(* ========================================================= *)
(*    FUN: HLI_ChannelModeReference                          *)
(* --------------------------------------------------------- *)
(*   Desc: switch channel to Reference mode / xxx            *)
(*   Author: MK, MiB, TV                                     *)
(*   Date: 03.03.2017                                        *)
(*   Rev.: 1.5                                               *)
(* ========================================================= *)


(************************************************************
	RefPosString:
	Element: parameter ( ASCII char set, Länge:256 Zeichen)

	Vorgabe zur Parametrierung der Referenzpunktfahrt.

	Ist dieser STRING leer, so wird defaultmäßig das
	Automatikprogramm "rpf.nc" angewählt.

	Ansonsten kann durch explizite Angabe der Achsen und
	Zeitpunkt im Format "G74
	<Achsbezeichner_1><Zeitpunkt_1> ...
	<Achsbezeichner_n><Zeitpunkt_n>"
	eine individuelle Referenzpunktfahrt vorgegeben werden.
*************************************************************)

IF (NOT gpCh[nChanIdx]^.channel_mc_control.mode_and_state.command_semaphor_rw) THEN  (* only if semaphor is FALSE...... *)
	IF stCmdModesStates.stStates.Selected THEN
		stCmdModesStates.stStates.Selected := FALSE;
		gpCh[nChanIdx]^.channel_mc_control.mode_and_state.command_w.to_mode := HLI_IMCM_REFERENCE_MODE;
		gpCh[nChanIdx]^.channel_mc_control.mode_and_state.command_w.to_state := HLI_IMCM_PROCESS_SELECTED;		
		gpCh[nChanIdx]^.channel_mc_control.mode_and_state.command_semaphor_rw := TRUE;	
	END_IF
	
	IF stCmdModesStates.stStates.Ready THEN
		stCmdModesStates.stStates.Ready := FALSE;
		gpCh[nChanIdx]^.channel_mc_control.mode_and_state.command_w.to_mode := HLI_IMCM_REFERENCE_MODE;
		gpCh[nChanIdx]^.channel_mc_control.mode_and_state.command_w.to_state := HLI_IMCM_PROCESS_READY;		
		pString := ADR(gpCh[nChanIdx]^.channel_mc_control.mode_and_state.command_w.parameter);	
		gpCh[nChanIdx]^.channel_mc_control.mode_and_state.command_semaphor_rw := TRUE;		
	END_IF
	
	IF stCmdModesStates.stStates.Active THEN
		stCmdModesStates.stStates.Active := FALSE;
		gpCh[nChanIdx]^.channel_mc_control.mode_and_state.command_w.to_mode := HLI_IMCM_REFERENCE_MODE;
		gpCh[nChanIdx]^.channel_mc_control.mode_and_state.command_w.to_state := HLI_IMCM_PROCESS_ACTIVE;		
		pString := ADR(gpCh[nChanIdx]^.channel_mc_control.mode_and_state.command_w.parameter);	
		pString^ := sRefPosString;
		gpCh[nChanIdx]^.channel_mc_control.mode_and_state.command_semaphor_rw:= TRUE;		
	END_IF
	
	IF stCmdModesStates.stStates.Hold THEN
		stCmdModesStates.stStates.Hold := FALSE;
		gpCh[nChanIdx]^.channel_mc_control.mode_and_state.command_w.to_mode := HLI_IMCM_REFERENCE_MODE;
		gpCh[nChanIdx]^.channel_mc_control.mode_and_state.command_w.to_state := HLI_IMCM_PROCESS_HOLD;		
		gpCh[nChanIdx]^.channel_mc_control.mode_and_state.command_semaphor_rw := TRUE;		
	END_IF
	
	IF stCmdModesStates.stStates.Reset THEN
		stCmdModesStates.stStates.Reset := FALSE;
		gpCh[nChanIdx]^.channel_mc_control.mode_and_state.command_w.to_mode:= HLI_IMCM_REFERENCE_MODE;
		gpCh[nChanIdx]^.channel_mc_control.mode_and_state.command_w.to_state := HLI_IMCM_PROCESS_DESELECTED;		
		gpCh[nChanIdx]^.channel_mc_control.mode_and_state.command_semaphor_rw := TRUE;		
	END_IF

	HLI3_ChannelModeReference := TRUE;
ELSE
	HLI3_ChannelModeReference := FALSE;
END_IF

END_FUNCTION

// CNC/2 OperationMode/HLI3_ChannelModeStandby
FUNCTION HLI3_ChannelModeStandby : BOOL
VAR_INPUT	 
	nChanIdx: INT;
	ProgramName: STRING(HLI_IMCM_MODE_STATE_PARAM_STRL);			
END_VAR

VAR_IN_OUT
	stCmdModesStates    : ST_CNCCmdModesStates;	
END_VAR

VAR
	pString: POINTER TO STRING(HLI_IMCM_MODE_STATE_PARAM_STRL);
	nCHan: INT;
END_VAR

(* ========================================================= *)
(*    FUN: HLI_ChannelModeStandby                            *)
(* --------------------------------------------------------- *)
(*   Desc: switch channel to Standby mode / xxx              *)
(*   Author: MK, MiB, TV                                     *)
(*   Date: 03.03.2017                                        *)
(*   Rev.: 1.5                                               *)
(* ========================================================= *)

IF (NOT gpCh[nChanIdx]^.channel_mc_control.mode_and_state.command_semaphor_rw) THEN  (* only if semaphor is FALSE...... *)
	IF stCmdModesStates.stStates.Selected THEN
		stCmdModesStates.stStates.Selected := FALSE;
		gpCh[nChanIdx]^.channel_mc_control.mode_and_state.command_w.to_mode := HLI_IMCM_STANDBY_MODE;
		gpCh[nChanIdx]^.channel_mc_control.mode_and_state.command_w.to_state := HLI_IMCM_PROCESS_SELECTED;
		pString := ADR(gpCh[nChanIdx]^.channel_mc_control.mode_and_state.command_w.parameter);			
		pString^ := ProgramName;				
		gpCh[nChanIdx]^.channel_mc_control.mode_and_state.command_semaphor_rw := TRUE;		
	END_IF
	
	IF stCmdModesStates.stStates.Ready THEN
		stCmdModesStates.stStates.Ready := FALSE;
		gpCh[nChanIdx]^.channel_mc_control.mode_and_state.command_w.to_mode := HLI_IMCM_STANDBY_MODE;
		gpCh[nChanIdx]^.channel_mc_control.mode_and_state.command_w.to_state := HLI_IMCM_PROCESS_READY;		
		pString := ADR(gpCh[nChanIdx]^.channel_mc_control.mode_and_state.command_w.parameter);			
		pString^ := ProgramName;	
		gpCh[nChanIdx]^.channel_mc_control.mode_and_state.command_semaphor_rw := TRUE;		
	END_IF
	
	IF stCmdModesStates.stStates.Active THEN
		stCmdModesStates.stStates.Active := FALSE;
		gpCh[nChanIdx]^.channel_mc_control.mode_and_state.command_w.to_mode := HLI_IMCM_STANDBY_MODE;
		gpCh[nChanIdx]^.channel_mc_control.mode_and_state.command_w.to_state := HLI_IMCM_PROCESS_ACTIVE;		
		pString := ADR(gpCh[nChanIdx]^.channel_mc_control.mode_and_state.command_w.parameter);			
		pString^ := ProgramName;	
		gpCh[nChanIdx]^.channel_mc_control.mode_and_state.command_semaphor_rw := TRUE;		
	END_IF
	
	IF stCmdModesStates.stStates.Hold THEN
		stCmdModesStates.stStates.Hold := FALSE;
		gpCh[nChanIdx]^.channel_mc_control.mode_and_state.command_w.to_mode := HLI_IMCM_STANDBY_MODE;
		gpCh[nChanIdx]^.channel_mc_control.mode_and_state.command_w.to_state:= HLI_IMCM_PROCESS_HOLD;		
		gpCh[nChanIdx]^.channel_mc_control.mode_and_state.command_semaphor_rw := TRUE;	
	END_IF
	
	IF stCmdModesStates.stStates.Reset THEN
		stCmdModesStates.stStates.Reset := FALSE;
		gpCh[nChanIdx]^.channel_mc_control.mode_and_state.command_w.to_mode := HLI_IMCM_STANDBY_MODE;
		gpCh[nChanIdx]^.channel_mc_control.mode_and_state.command_w.to_state:= HLI_IMCM_PROCESS_DESELECTED;		
		gpCh[nChanIdx]^.channel_mc_control.mode_and_state.command_semaphor_rw := TRUE;		
	END_IF
	
	HLI3_ChannelModeStandby := TRUE;
ELSE
	HLI3_ChannelModeStandby := FALSE;
END_IF

END_FUNCTION

// CNC/2 OperationMode/HLI3_ChannelReset
FUNCTION HLI3_ChannelReset : BOOL
VAR_INPUT
	/// Channel index 
	nChanIdx: INT;
END_VAR
VAR
	/// local pointer to Data of actual Channel 
	pChannelData: POINTER TO HIGH_LEVEL_INTERFACE_CH;
END_VAR

(* ========================================================= *)
(*    FUN: HLI_ChannelReset                                  *)
(* --------------------------------------------------------- *)
(*   Desc:                                                   *)
(* Author: MK ,MiB, TV                                       *)
(*   Date: 17.01.2018                                        *)
(*   Rev.: 1.1                                               *)
(* ========================================================= *)

HLI3_ChannelReset := FALSE;
IF NOT HLI3_CheckChannelValid(nChannel := nChanIdx) THEN
	RETURN;
END_IF

(* get pointer to channel data *)
pChannelData := gpCh[nChanIdx];
IF (pChannelData = 0) THEN   (* check for zero pointer *)
	RETURN;
END_IF

(* is a reset commanded *)
IF pChannelData^.bahn_lc_control.plc_reset.command_r = TRUE THEN
	
(* Reset all M- and H-Functions whenn the channel gets resetted *)
	HLI3_ChannelResetMFunctions(nChanIdx);
	HLI3_ChannelResetHFunctions(nChanIdx);
	
	(* quit this reset *)
	pChannelData^.bahn_lc_control.plc_reset.state_w := TRUE;	
	HLI3_ChannelReset := TRUE;
END_IF

END_FUNCTION

// CNC/4 MHT-Function/HLI3_ChannelResetMFunctions
FUNCTION HLI3_ChannelResetMFunctions : BOOL
VAR_INPUT
	/// Channel number 
	nChanIdx: INT;
END_VAR
VAR
	idx: INT;
END_VAR

(* ========================================================= *)
(*    FUN: HLI_ChannelResetMFunctions                        *)
(* --------------------------------------------------------- *)
(*   Desc:                                                   *)
(* Author: MK                                                *)
(*   Date: 10.05.2007                                        *)
(*   Rev.: 1.00                                              *)
(* ========================================================= *)

IF NOT HLI3_CheckChannelValid(nChannel := nChanIdx) THEN
	HLI3_ChannelResetMFunctions := FALSE;
	RETURN; (* A b b r u c h *)
END_IF


FOR idx := 1 TO 999 DO
	CNCSystem.Channel[nChanIdx].M[idx].bState_rw := FALSE;
	CNCSystem.Channel[nChanIdx].M[idx].bRes := FALSE;
	CNCSystem.Channel[nChanIdx].actM_r :='';
END_FOR

HLI3_ChannelResetMFunctions := TRUE;

END_FUNCTION

// CNC/4 MHT-Function/HLI3_ChannelResetHFunctions
FUNCTION HLI3_ChannelResetHFunctions : BOOL
VAR_INPUT
	/// Channel number 
	nChanIdx: INT;
END_VAR
VAR
	idx: INT;
END_VAR

(* ========================================================= *)
(*    FUN: HLI_ChannelResetHFunctions                        *)
(* --------------------------------------------------------- *)
(*   Desc:                                                   *)
(* Author: MiB                                                *)
(*   Date: 23.11.2012                                        *)
(*   Rev.: 1.1                                              *)
(* ========================================================= *)



IF NOT HLI3_CheckChannelValid(nChannel := nChanIdx) THEN
	HLI3_ChannelResetHFunctions := FALSE;
	RETURN; (* A b b r u c h *)
END_IF


FOR idx := 0 TO 999 DO
	CNCSystem.Channel[nChanIdx].H[idx].bState_rw := FALSE;
	CNCSystem.Channel[nChanIdx].H[idx].bRes := FALSE;
	CNCSystem.Channel[nChanIdx].actH_r :='';
END_FOR

HLI3_ChannelResetHFunctions := TRUE;

END_FUNCTION

// CNC/2 OperationMode/HLI3_ChannelResetRequest
FUNCTION_BLOCK HLI3_ChannelResetRequest
VAR_INPUT
	bExec: BOOL;
	/// Channel number 
	nChanIdx: INT;
	pChannel: POINTER TO ST_CncChannel;
END_VAR
VAR_OUTPUT
	bBusy: BOOL;
	bSwitchMode: BOOL;
	nMode: UDINT;
END_VAR
VAR
	fbRtrigExec: R_TRIG;
	/// Index of channel specific HLI area 
	nHliChIfcIdx: INT;
	nState: UINT;
	pCommand: POINTER TO HLI_PROC_TRANS_TO_MODE_STATE;
	actualMode: UDINT;
	fbTON: TON;
END_VAR

(******************************************************************************)
(* POU:				HLI_ChannelResetRequest									*)
(* Type:				Function block										*)
(* Customer:		Common													*)
(* Date:				07/11/16											*)
(* Last:				10/03/10											*)
(* -------------------------------------------------------------------------- *)
(* Revision:		1.0														*)
(* Author:			MiB														*)
(* Description: 	Performs a reset in the given cnc channel. 				*)
(* -------------------------------------------------------------------------- *)
(* Revision:		1.10													*)
(* Author:			MiB														*)
(* Description: 	Changed from PRG to FB.									*)
(* -------------------------------------------------------------------------- *)
(* Revision:		2.00															*)
(* Author:			HR																*)
(* Description: 	Deleted references to global variable 'PLCMachineMode[n]'.		*)
(*						The FB now works with VAR_OUTPUT 'nMode' and 'bSwitchMode'	*)
(*						as a callback to the initiator to let it perform the change	*)
(*						of the operation mode by itself in order to reset the cnc	*)
(*						channel.													*)
(* -------------------------------------------------------------------------- *)
(* Revision:		2.01																			*)
(* Author:			TV																				*)
(* Description: 	Expand State "Wait for previous mode"  *)
(*				Prevent to trigger the state machine during the mode switch							*)
(* -------------------------------------------------------------------------- *)
(* Revision:		2.02																			*)
(* Author:			MiB																				*)
(* Description: 	Tc3*)
(******************************************************************************)


fbRtrigExec( clk := bExec   );

IF fbRtrigExec.Q THEN
	bBusy := TRUE;
	nState := 10;
END_IF


CASE nState OF

0:		(* IDLE *)
		bBusy := FALSE;

10:	(* Reset request: get actual opmode *)
		bSwitchMode := FALSE;
		actualMode := gpCh[nChanIdx]^.channel_mc_control.mode_and_state.state_r.mode;
		nState := nState + 10;

20:  (* switch to standby *)
		bSwitchMode := TRUE;
		nMode:= HLI_IMCM_STANDBY_MODE;
		fbTON(IN:= FALSE);
		nState := nState + 10;

30: 	(* Wait for modeswitch *)
		bSwitchMode := FALSE;
		fbTON(IN:= TRUE, PT:= t#2000ms);
	 	IF gpCh[nChanIdx]^.channel_mc_control.mode_and_state.state_r.mode = HLI_IMCM_STANDBY_MODE THEN
			nState := nState + 10;
		END_IF
		IF fbTON.Q THEN
			(* Timeout Error -> go on with next step *)
			nState := nState + 10;
		END_IF

40:	(* switch back to previous mode *)
		bSwitchMode := TRUE;
		nMode:= actualMode;
		fbTON(IN:= FALSE);
		nState := nState + 10;

50:	(* Wait for previous mode  *)
		fbTON(IN:= TRUE, PT:= t#2000ms);
		IF (gpCh[nChanIdx]^.channel_mc_control.mode_and_state.state_r.mode = 	actualMode) THEN
			nState := nState + 10;
		END_IF
		IF fbTON.Q THEN
			(* Timeout Error -> go on with next step *)
			nState := nState + 10;
		END_IF

60: 	(* ready *)
		bSwitchMode := FALSE;
		nState := 0;

END_CASE



(* das muss ins aufrufende Programm: (HLI_CNCChannel)

VAR
	bResetRequest:			BOOL;
	fbRTrigReset:			R_TRIG;
	ChannelResetRequest: HLI_ChannelResetRequest;
END_VAR

fbRTrigReset(clk := bStateReset);
IF fbRTrigReset.Q THEN
	bResetRequest := TRUE;
	...
END_IF

(* Handle Channel reset *)
ChannelResetRequest
	(bExec 		:= bResetRequest ,
	 nChan 		:= nChan,
	 pChannel	:= ADR(CNCSystem.Channel[nChan])
	);

IF ChannelResetRequest.bSwitchMode THEN
	bModeStandby	:= bModeStandby OR (ChannelResetRequest.nMode = HLI_IMCM_STANDBY_MODE);
	bModeAutomatic	:= bModeAutomatic OR (ChannelResetRequest.nMode = HLI_IMCM_AUTOMATIC_MODE);
	bModeManual		:= bModeManual OR (ChannelResetRequest.nMode = HLI_IMCM_MANUAL_MODE);
	bModeMDI			:= bModeMDI OR (ChannelResetRequest.nMode = HLI_IMCM_MDI_MODE);
	bModeReference	:= bModeReference OR (ChannelResetRequest.nMode = HLI_IMCM_REFERENCE_MODE);
END_IF

IF bResetRequest AND NOT ChannelResetRequest.bBusy THEN
	bResetRequest := FALSE;
END_IF

*)

END_FUNCTION_BLOCK

// CNC/2 OperationMode/HLI3_CNCChannel
FUNCTION_BLOCK HLI3_CNCChannel
VAR_INPUT
	/// index of channel
	nChanIdx: INT;
 
	bCmdAutomatic : BOOL;
	bCmdManual : BOOL;
    bCmdReference : BOOL;
    bCmdMDI : BOOL;		
	bCmdStart : BOOL;
	bCmdStop  : BOOL;
	bCmdReset : BOOL;		
	/// must be xxx.nc 
	sProgramName: STRING(HLI_IMCM_MODE_STATE_PARAM_STRL);
	/// the MDI string 
	sMDIString: STRING(HLI_IMCM_MODE_STATE_PARAM_STRL);
	/// static signal 
	bBackwardMotion: BOOL;
	/// static signal 
	bFeedHold: BOOL;
	/// static signal 
	bReducedFeed: BOOL;
	/// static signal 
	bSingleBlock: BOOL;
	/// static signal 
	bPrgBlockIgnore: BOOL;
	/// static signal 
	bM01Stop: BOOL;
	/// static signal 
	nSyntaxCheck: DINT;		
	// Manual Mode
	stManualModeParameter: ST_ManualModeParameter;
	stManualModeControlElements: ST_ManualModeControlElements;
	// M30 Acknowledgement inside Channel FB
	bM30Acknowledgement : BOOL;
	// Override 
	nFeedOverride : UINT;
	nRapidFeedOverride : UINT;
	bEmergencyStop : BOOL;
	stOptions : ST_CNC_CH_Options;
END_VAR
VAR_IN_OUT
	/// please only a flank 
	bModeStandby: BOOL;
	/// please only a flank 
	bModeAutomatic: BOOL;
	/// please only a flank 
	bModeManual: BOOL;
	/// please only a flank 
	bModeMDI: BOOL;
	/// please only a flank 
	bModeReference: BOOL;
	/// please only a flank 
	bStateSelect: BOOL;
	/// please only a flank 
	bStateReady: BOOL;
	/// please only a flank 
	bStateStart: BOOL;
	/// please only a flank 
	bStateStop: BOOL;
	/// please only a flank 
	bStateReset: BOOL;
	/// please only a flank 
	bDoSingleBlock: BOOL;
	// manual mode
	stManualModeControlElementState: ST_ManualModeControlElementState;
END_VAR
VAR
	bGoToActive	: BOOL;	 	
	/// Pointer to channel control structure 
	pChannel: POINTER TO ST_CncChannel;
	ChannelMHTFunction: HLI3_QuitChannelMHTFunction;
	/// Current Mode of Operation Modes;
	currentMode: UDINT;
	/// Current State of Operation Modes;
	currentState: UDINT;
	idx: INT;	
	bCheckOpModeFirst: BOOL;
	fbRTrigReset: R_TRIG;
	bResetRequest: BOOL;
	ChannelResetRequest: HLI3_ChannelResetRequest;
	nChan: INT;
	nStateAutoMDIStart: INT;
	ModeManual : HLI3_ManualModeHandler;	
	stCmdModesStates    : ST_CNCCmdModesStates;

	fbRTrigCmdStart: R_TRIG;
	fbRTrigCmdStop:  R_TRIG;
	fbRTrigCmdReset: R_TRIG;	
	fbRTrigCmdAutomatic : R_TRIG;
	fbRTrigCmdManual : R_TRIG;
    fbRTrigCmdReference : R_TRIG;
    fbRTrigCmdMDI : R_TRIG;		
END_VAR

(* ========================================================= *)
(*     FB: HLI_CNCChannel                                    *)
(* --------------------------------------------------------- *)
(*   Desc:                                                   *)
(*   Author: MK ,MiB, TV, Rch                                *)
(*   Date: 2018.03.29                                        *)
(*   Rev.: 1.15                                               *)
(*         1.2 Before "start" the state is swicthed to 		 *)
(*				"Selected" and "Ready" to ensure that the    *)	
(*				actual selected program will start 			 *)
(*		   1.3  BugFix : nChanNo at HLI3_ChannelModeMDI()    *)
(*         1.4  Implement state switch to "selected" and "ready"  *)         
(*		   1.5  Channel reset via commanding state 			 *)
(*              RESETTING directly							 *)  
(*		   1.6  Optimized Channel reset via commanding state *)
(*				RESETTING directly						     *)
(*		   1.7  Init Paramerer for Manual mode as input parameter*)
(*		   1.8  BugFix : max index for HLI3_AxisReset		*)
(*		   1.9  Implementation of HLI3_ManualModeHandler	*)
(*		   1.10 Implementation of Input bM30Acknowledgement	*)
(*		   1.12 Optimized Operating modes					*)
(*		   1.13 Optimized Operating modes				    *)
(*		   1.14 Optimized M and H Function during Reset     *)
(*		   1.15 Implementation of ST_CNC_CH_Options Structure *)
(* =========================================================*)

IF NOT HLI3_CheckChannelValid(nChannel := nChanIdx) THEN
	RETURN;
END_IF

(* handle reset request *)
fbRTrigReset
	(CLK := bStateReset);
	
IF fbRTrigReset.Q THEN
	nStateAutoMDIStart := 0;
	CNCSystem.Channel[nChanIdx].ToolData.bOldToolDataExist := FALSE;
	CNCSystem.Channel[nChanIdx].ToolData.bToolRequest := FALSE;
	CNCSystem.Channel[nChanIdx].ToolData.bResetToolRequest := TRUE;
END_IF

fbRTrigCmdAutomatic(CLK:=bCmdAutomatic);
fbRTrigCmdManual(CLK:=bCmdManual);
fbRTrigCmdReference(CLK:=bCmdReference);
fbRTrigCmdMDI(CLK:=bCmdMDI);	

fbRTrigCmdStart(CLK:=bCmdStart);  
fbRTrigCmdStop(CLK:=bCmdStop);
fbRTrigCmdReset(CLK:=bCmdReset);

(* ************************************* *)
(*  Motion-Control                       *)
(* ************************************* *)

(* EmergencyStop *)
HLI3_ChannelSetEmergencyStop(nChanIdx:=nChanIdx, bEStop := bEmergencyStop);
 
(* Feed Override [0.1%] *)
HLI3_SetChannelOverride(nChanIdx:=nChanIdx, nOverride := nFeedOverride);

(* Rapid feed override [0.1%], must be activated with parameter P-CHAN-00181 *)
HLI3_SetChannelRapidOverride(nChanIdx:=nChanIdx, nOverride := nRapidFeedOverride);

(* Backward Motion *)
HLI3_ChannelSetBackwardMotion(nChanIdx:=nChanIdx, bBackwardMotion:=bBackwardMotion);

(* Program Block Ignore *)
HLI3_ChannelSetProgramBlockIgnore(nChanIdx:=nChanIdx, bPrgBlockIgnore:=bPrgBlockIgnore);

(* Feed Hold *)
HLI3_ChannelSetFeedHold(nChanIdx:=nChanIdx, bFeedHold:=bFeedHold);

(* Single Step *)
HLI3_ChannelSetSingleBlock(nChanIdx:=nChanIdx, bSingleBlock:=bSingleBlock);

(* Reduced Feed *)
HLI3_ChannelSetReducedFeed(nChanIdx:=nChanIdx, bReducedFeed:=bReducedFeed);

(* Syntax Check *)
gpCh[nChanIdx]^.decoder_mc_control.execution_mode.command_w := nSyntaxCheck;

(* Optional stop M01 *)
gpCh[nChanIdx]^.bahn_mc_control.m01_stop_enable.command_w := bM01Stop;


(* ************************************ *)
(*  MHT-Function                        *)
(* ************************************ *)

(* MHT-Function, channel *)
ChannelMHTFunction(nChanIdx:=nChanIdx, bM30Acknowledgement := bM30Acknowledgement);

(* ************************************* *)
(*  Channel Status Info and error        *)
(* ************************************* *)
HLI3_GetChannelStatusInfo(nChanIdx:=nChanIdx);
HLI3_GetChannelError(nChanIdx:=nChanIdx);

(* ************************************* *)
(*  do single stepping                   *)
(* ************************************* *)
(* Achtung: hier noch anpassen, nur in Abhaengigkeit vom aktuellen Status den Start setzen *)
IF bDoSingleBlock THEN
	bDoSingleBlock := FALSE;
	bStateStart 	:= TRUE;
END_IF

(* ************************************* *)
(*  Operation Modes                      *)
(* ************************************* *)
(* Target modes and states *)
pChannel := ADR(CNCSystem.Channel[nChanIdx]);
OpModes();

(* OperationMode Standby *)
IF stCmdModesStates.stModes.Standby = TRUE THEN
	HLI3_ChannelModeStandby(nChanIdx := nChanIdx,ProgramName:=sProgramName, stCmdModesStates:=stCmdModesStates);
END_IF

(* OperationMode Auto *)
IF stCmdModesStates.stModes.Auto = TRUE THEN
	HLI3_ChannelModeAuto(nChanIdx := nChanIdx, ProgramName:=sProgramName, stCmdModesStates:=stCmdModesStates );
END_IF

(* OperationMode MDI *)
IF stCmdModesStates.stModes.MDI THEN
	(*sProgramName := PLCCncMDIString;*)
	HLI3_ChannelModeMDI(nChanIdx := nChanIdx, pMDIString:=ADR(sMDIString),stCmdModesStates:=stCmdModesStates);
END_IF

(* OperationMode Reference *)
IF stCmdModesStates.stModes.Homing THEN
	sProgramName := '';	(* we choose the default program: rpf.nc *)
	HLI3_ChannelModeReference(nChanIdx := nChanIdx, sRefPosString:=sProgramName, stCmdModesStates:=stCmdModesStates);
END_IF

(* OperationMode Manual *)
IF stCmdModesStates.stModes.Manual THEN	
	HLI3_ChannelModeManual(nChanIdx := nChanIdx, stCmdModesStates:=stCmdModesStates);
END_IF

ModeManual
	(stManualModeParameter  	 	 := stManualModeParameter,
	 stManualModeControlElements	 := stManualModeControlElements,
	 stManualModeControlElementState := stManualModeControlElementState,
	 stCmdModesStates				 := stCmdModesStates,  	
	 arrAxisInG201 				      => stManualModeState[nChan].arrAxisInG201
);
			
(* Reset *)
HLI3_ChannelReset(nChanIdx:=nChanIdx);							(* channel *)
FOR idx := 0 TO UDINT_TO_INT(gNrAx-1) DO							(* axis *)
	HLI3_AxisReset(nChanNo:=nChanIdx+1, nHliAxisIdx:=idx);
END_FOR

ACTION AutoMDIStart:



CASE nStateAutoMDIStart OF
	0:		;(* IDLE *)
	
	10: (* swicth to selected *)
		stCmdModesStates.stStates.Selected := TRUE;
		nStateAutoMDIStart := nStateAutoMDIStart +10;
		
	20: (* wait for selected *)
		IF (pChannel^.ActState =  HLI_IMCM_PROCESS_SELECTED) THEN
			stCmdModesStates.stStates.Ready := TRUE;
			nStateAutoMDIStart := nStateAutoMDIStart +10;
		END_IF
	30: (* Wait for ready and then start*)
		IF (pChannel^.ActState =  HLI_IMCM_PROCESS_READY) THEN
			stCmdModesStates.stStates.Active := TRUE; 
			nStateAutoMDIStart := 0;
		END_IF
	
END_CASE
END_ACTION

ACTION OpModes:
(*************************************************)
(* Restore internal state at first run           *)
(* after PLC reset                               *)
(*************************************************)

IF bCheckOpModeFirst = FALSE THEN
	bCheckOpModeFirst := TRUE;
	currentMode := HLI3_GetChannelMode(nChanIdx:=nChanIdx);
	IF currentMode = HLI_IMCM_STANDBY_MODE THEN
		stCmdModesStates.stModes.Standby := TRUE;
	END_IF
	IF currentMode = HLI_IMCM_AUTOMATIC_MODE THEN
		stCmdModesStates.stModes.Auto := TRUE;
	END_IF
	IF currentMode = HLI_IMCM_MDI_MODE THEN
		stCmdModesStates.stModes.MDI := TRUE;
	END_IF
	IF currentMode = HLI_IMCM_MANUAL_MODE THEN
		stCmdModesStates.stModes.Manual := TRUE;
	END_IF
	IF currentMode = HLI_IMCM_REFERENCE_MODE THEN		
		stCmdModesStates.stModes.Homing := TRUE;
	END_IF
END_IF


(*************************************************)
(* Operation Modes                               *)
(*************************************************)

IF bModeStandby THEN
	bModeStandby := FALSE;
	stCmdModesStates.stModes.Standby		:= TRUE;
	stCmdModesStates.stModes.Auto			:= FALSE;
	stCmdModesStates.stModes.MDI			:= FALSE;
	stCmdModesStates.stModes.Manual		:= FALSE;
	stCmdModesStates.stModes.Homing		:= FALSE;


	stCmdModesStates.stStates.Selected	:= TRUE;
END_IF

IF bModeAutomatic OR fbRTrigCmdAutomatic.Q THEN
	bModeAutomatic 				:= FALSE;
	bGoToActive					:= FALSE;
	stCmdModesStates.stModes.Standby		:= FALSE;
	stCmdModesStates.stModes.Auto			:= TRUE;
	stCmdModesStates.stModes.MDI			:= FALSE;
	stCmdModesStates.stModes.Manual		:= FALSE;
	stCmdModesStates.stModes.Homing		:= FALSE;

	stCmdModesStates.stStates.Selected	:= TRUE;
END_IF

IF bModeMDI OR fbRTrigCmdMDI.Q THEN
	bModeMDI := FALSE;
	bGoToActive					:= FALSE;
	stCmdModesStates.stModes.Standby		:= FALSE;
	stCmdModesStates.stModes.Auto			:= FALSE;
	stCmdModesStates.stModes.MDI			:= TRUE;
	stCmdModesStates.stModes.Manual		:= FALSE;
	stCmdModesStates.stModes.Homing		:= FALSE;

	stCmdModesStates.stStates.Selected	:= TRUE;
END_IF

IF bModeManual OR fbRTrigCmdManual.Q THEN
	bModeManual := FALSE;
	stCmdModesStates.stModes.Standby		:= FALSE;
	stCmdModesStates.stModes.Auto			:= FALSE;
	stCmdModesStates.stModes.MDI			:= FALSE;
	stCmdModesStates.stModes.Manual		:= TRUE;
	stCmdModesStates.stModes.Homing		:= FALSE;

	stCmdModesStates.stStates.Active		:= TRUE;
END_IF

IF bModeReference OR fbRTrigCmdReference.Q THEN
	bModeReference := FALSE;
	bGoToActive					:= FALSE;
	stCmdModesStates.stModes.Standby		:= FALSE;
	stCmdModesStates.stModes.Auto			:= FALSE;
	stCmdModesStates.stModes.MDI			:= FALSE;
	stCmdModesStates.stModes.Manual		:= FALSE;
	stCmdModesStates.stModes.Homing		:= TRUE;
	
	IF stOptions.bReferenceModeStartRequired THEN
		stCmdModesStates.stStates.Selected	:= TRUE;
	ELSE
		stCmdModesStates.stStates.Active	:= TRUE;			
	END_IF	
	
END_IF



(*************************************************)
(* Operation States                              *)
(*************************************************)

currentMode := HLI3_GetChannelMode(nChanIdx:=nChanIdx);
currentState := HLI3_GetChannelState(nChanIdx:=nChanIdx);

CASE currentMode OF
	(*-------------------------------------------------------------------*)
	HLI_IMCM_STANDBY_MODE:
		IF bStateReset OR fbRTrigReset.Q THEN
			stCmdModesStates.stModes.Standby := TRUE;
			stCmdModesStates.stStates.Reset := TRUE;
		END_IF

	(*-------------------------------------------------------------------*)
	HLI_IMCM_AUTOMATIC_MODE:
		IF bStateStart OR fbRTrigCmdStart.Q THEN  (* replaced a simple 'start' by a sequence which switches the state to selected and ready*)
			IF currentState <> HLI_IMCM_PROCESS_HOLD AND currentState <> HLI_IMCM_PROCESS_ACTIVE THEN
				nStateAutoMDIStart := 10;
			ELSE
				stCmdModesStates.stStates.Active := TRUE; 
			END_IF					   	
		END_IF
		IF nStateAutoMDIStart <> 0 THEN
			AutoMDIStart();
		END_IF

		IF (bStateStop OR fbRTrigCmdStop.Q) AND currentState <> HLI_IMCM_PROCESS_DESELECTED THEN
			stCmdModesStates.stStates.Hold := TRUE;
		END_IF

		IF bStateReady THEN
			stCmdModesStates.stStates.Ready := TRUE;
		END_IF

		IF bStateReset OR fbRTrigCmdReset.Q THEN
			stCmdModesStates.stStates.Reset := TRUE;
			CNCSystem.Channel[nChanIdx].ToolData.bOldToolDataExist := FALSE;
			CNCSystem.Channel[nChanIdx].ToolData.bToolRequest := FALSE;
			CNCSystem.Channel[nChanIdx].ToolData.bResetToolRequest := TRUE;			
		END_IF
		
		IF bStateSelect THEN
			stCmdModesStates.stStates.Selected := TRUE;
		END_IF		

	(*-------------------------------------------------------------------*)
	HLI_IMCM_MDI_MODE:
		IF bStateStart OR fbRTrigCmdStart.Q THEN
			IF currentState <> HLI_IMCM_PROCESS_HOLD AND currentState <> HLI_IMCM_PROCESS_ACTIVE THEN
				nStateAutoMDIStart := 10;
			ELSE
				stCmdModesStates.stStates.Active := TRUE; 
			END_IF
		END_IF
		
		IF nStateAutoMDIStart <> 0 THEN
			AutoMDIStart();
		END_IF
		
		IF (bStateStop OR fbRTrigCmdStop.Q) AND currentState <> HLI_IMCM_PROCESS_DESELECTED THEN
			stCmdModesStates.stStates.Hold := TRUE;
		END_IF

		IF bStateSelect THEN
			stCmdModesStates.stStates.Selected := TRUE;
		END_IF
		
		IF bStateReady THEN
			stCmdModesStates.stStates.Ready := TRUE;
		END_IF

		IF bStateReset OR fbRTrigCmdReset.Q THEN
			stCmdModesStates.stStates.Reset := TRUE;
			CNCSystem.Channel[nChanIdx].ToolData.bOldToolDataExist := FALSE;
			CNCSystem.Channel[nChanIdx].ToolData.bToolRequest := FALSE;
			CNCSystem.Channel[nChanIdx].ToolData.bResetToolRequest := TRUE;			
		END_IF

	(*-------------------------------------------------------------------*)
	HLI_IMCM_MANUAL_MODE:
		IF bStateStart OR fbRTrigCmdStart.Q OR ((currentState = HLI_IMCM_PROCESS_SELECTED) AND bGoToActive) THEN
			bGoToActive := FALSE;	
			stCmdModesStates.stStates.Active 	:= TRUE;
		END_IF

		IF bStateReady THEN
			stCmdModesStates.stStates.Ready 	:= TRUE;
		END_IF

		IF bStateSelect THEN
			stCmdModesStates.stStates.Selected := TRUE;
		END_IF

		IF bStateStop OR fbRTrigCmdStop.Q THEN
			stCmdModesStates.stStates.Hold := TRUE;
		END_IF

		IF (bStateReset OR fbRTrigCmdReset.Q) THEN	
			CNCSystem.Channel[nChanIdx].ToolData.bOldToolDataExist := FALSE;
			CNCSystem.Channel[nChanIdx].ToolData.bToolRequest := FALSE;
			CNCSystem.Channel[nChanIdx].ToolData.bResetToolRequest := TRUE;
			
			stCmdModesStates.stStates.Reset := TRUE;
			IF stCmdModesStates.stModes.Manual THEN
				bGoToActive := TRUE;
			END_IF
		END_IF

	(*-------------------------------------------------------------------*)
	HLI_IMCM_REFERENCE_MODE:
		IF bStateStart OR fbRTrigCmdStart.Q THEN
			stCmdModesStates.stStates.Active := TRUE;
		END_IF

		IF bStateStop OR fbRTrigCmdStop.Q THEN
			stCmdModesStates.stStates.Hold := TRUE;
		END_IF

		IF bStateReset OR fbRTrigCmdReset.Q THEN
			CNCSystem.Channel[nChanIdx].ToolData.bOldToolDataExist := FALSE;
			CNCSystem.Channel[nChanIdx].ToolData.bToolRequest := FALSE;
			CNCSystem.Channel[nChanIdx].ToolData.bResetToolRequest := TRUE;			
			stCmdModesStates.stStates.Reset := TRUE;
		END_IF
END_CASE


bStateStart 	:= FALSE;
bStateStop 		:= FALSE;
bStateReset 	:= FALSE;
bStateSelect 	:= FALSE;
bStateready 	:= FALSE;
END_ACTION

END_FUNCTION_BLOCK

// CNC/3 Control/HLI3_ChannelSetEmergencyStop
FUNCTION HLI3_ChannelSetEmergencyStop : BOOL
VAR_INPUT
	/// Number of channel 
	nChanIdx: INT;
	bEStop: BOOL;
END_VAR

(****************************************************************************************)
(* POU:			HLI_ChannelSetEmergenyStop												*)
(* Type:		Function block															*)
(* Customer:	Common																	*)
(* Date:		09/03/12																*)
(* Last:		20/11/12																*)
(* ------------------------------------------------------------------------------------ *)
(* Revision:	1.0																		*)
(* Author:		HR,MiB																	*)
(* Description: (Re-)Sets the channel specific emergency stop unit.						*)
(****************************************************************************************)

HLI3_ChannelSetEmergencyStop := FALSE;
IF NOT HLI3_CheckChannelValid(nChannel := nChanIdx) THEN
	RETURN;
END_IF

(* if the stop button from the HMI is selected the request is set *)
gpCh[nChanIdx]^.bahn_mc_control.emergency_stop.command_w := bEStop;

HLI3_ChannelSetEmergencyStop		:= TRUE;

END_FUNCTION

// CNC/3 Control/HLI3_SetChannelOverride
FUNCTION HLI3_SetChannelOverride : BOOL
VAR_INPUT
	/// Number of channel 
	nChanIdx: INT;
	nOverride: UINT;
END_VAR

(* ========================================================= *)
(*    FUN: HLI_SetChannelOverride                            *)
(* --------------------------------------------------------- *)
(*   Desc: Set the channel Override                          *)
(* Author: MK, MiB                                           *)
(*   Date: 20.11.2012                                        *)
(*   Rev.: 1.2  2017.10.25                                   *)
(* ========================================================= *)

IF NOT HLI3_CheckChannelValid(nChannel := nChanIdx) THEN
	HLI3_SetChannelOverride := FALSE;
	RETURN;
END_IF

(* Limit the override *)
IF nOverride > 2000 THEN nOverride := 2000; END_IF  // MiB 2017.10.25 valid maximum in cnc core is 2000
IF nOverride < 0 THEN nOverride := 0; END_IF

gpCh[nChanIdx]^.bahn_mc_control.override_feedrate.command_w := nOverride;

HLI3_SetChannelOverride := TRUE;

END_FUNCTION

// CNC/3 Control/HLI3_SetChannelRapidOverride
FUNCTION HLI3_SetChannelRapidOverride : BOOL
VAR_INPUT
	/// Number of channel 
	nChanIdx: INT;
	nOverride: UINT;
END_VAR

(* ========================================================= *)
(*    FUN: HLI_SetChannelRapidOverride                       *)
(* --------------------------------------------------------- *)
(*   Desc: Set the channel Override for rapid movements      *)
(*   Author: TV , MiB                                        *)
(*   Date: 07.02.2017                                        *)
(*   Rev.: 1.1                                               *)
(* ========================================================= *)

IF NOT HLI3_CheckChannelValid(nChannel := nChanIdx) THEN
	HLI3_SetChannelRapidOverride := FALSE;
	RETURN;
END_IF

(* Limit the override *)
IF nOverride > 1000	THEN nOverride := 1000; END_IF  // MiB 2017.10.25 maximum is 1000 (ref HLI manual)
IF nOverride < 0 THEN nOverride := 0; END_IF

gpCh[nChanIdx]^.bahn_mc_control.override_rapid_move.enable_w := TRUE;
gpCh[nChanIdx]^.bahn_mc_control.override_rapid_move.command_w := nOverride;

HLI3_SetChannelRapidOverride := TRUE;

END_FUNCTION

// CNC/3 Control/HLI3_ChannelSetBackwardMotion
FUNCTION HLI3_ChannelSetBackwardMotion : BOOL
VAR_INPUT
	/// Number of channel 
	nChanIdx: INT;
	bBackwardMotion: BOOL;
END_VAR

(* ========================================================= *)
(*    FUN: HLI_ChannelSetBackwardMotion                      *)
(* --------------------------------------------------------- *)
(*   Desc:                                                   *)
(* Author: MK, MiB                                           *)
(*   Date: 20.11.2012                                        *)
(*   Rev.: 1.1                                               *)
(* ========================================================= *)

HLI3_ChannelSetBackwardMotion := FALSE;
IF NOT HLI3_CheckChannelValid(nChannel := nChanIdx) THEN
	RETURN;
END_IF

gpCh[nChanIdx]^.bahn_mc_control.backward_motion.command_w := bBackwardMotion;

HLI3_ChannelSetBackwardMotion := TRUE;

END_FUNCTION

// CNC/3 Control/HLI3_ChannelSetProgramBlockIgnore
FUNCTION HLI3_ChannelSetProgramBlockIgnore : BOOL
VAR_INPUT
	/// Number of channel 
	nChanIdx: INT;
	bPrgBlockIgnore: BOOL;
END_VAR

(* ========================================================= *)
(*    FUN: HLI_SetProgramBlockIgnore                         *)
(* --------------------------------------------------------- *)
(*   Desc:                                                   *)
(* Author: MK, MiB , TV                                      *)
(*   Date: 20.12.2012                                        *)
(*   Last: 19.11.2013                                        *)
(*   Rev.: 1.0                                               *)
(* ========================================================= *)

HLI3_ChannelSetProgramBlockIgnore := FALSE;
IF NOT HLI3_CheckChannelValid(nChannel := nChanIdx) THEN
	RETURN;
END_IF

(* program block ignore *)
IF bPrgBlockIgnore THEN
	gpCh[nChanIdx]^.decoder_mc_control.program_block_ignore.command_w := 1;
ELSE
	gpCh[nChanIdx]^.decoder_mc_control.program_block_ignore.command_w := 0;
END_IF

HLI3_ChannelSetProgramBlockIgnore := TRUE;

END_FUNCTION

// CNC/3 Control/HLI3_ChannelSetFeedHold
FUNCTION HLI3_ChannelSetFeedHold : BOOL
VAR_INPUT
	/// Number of channel 
	nChanIdx: INT;
	bFeedHold: BOOL;
END_VAR

(* ========================================================= *)
(*    FUN: HLI_ChannelSetFeedHold                            *)
(* --------------------------------------------------------- *)
(*   Desc:                                                   *)
(* Author: MK , MiB                                          *)
(*   Date: 20.11.2012                                        *)
(*   Rev.: 1.1                                               *)
(* ========================================================= *)

HLI3_ChannelSetFeedHold := FALSE;
IF NOT HLI3_CheckChannelValid(nChannel := nChanIdx) THEN
	RETURN;
END_IF

(* if the stop button from the HMI is selected the request is set *)
gpCh[nChanIdx]^.bahn_mc_control.feedhold.command_w := bFeedHold OR gpCh[nChanIdx]^.bahn_mc_control.feedhold.request_r;
HLI3_ChannelSetFeedHold := TRUE;

END_FUNCTION

// CNC/3 Control/HLI3_ChannelSetSingleBlock
FUNCTION HLI3_ChannelSetSingleBlock : BOOL
VAR_INPUT
	/// Number of channel 
	nChanIdx: INT;
	bSingleBlock: BOOL;
END_VAR

(* ========================================================= *)
(*    FUN: HLI3_ChannelSetSingleBlock                        *)
(* --------------------------------------------------------- *)
(*   Desc:                                                   *)
(* Author: MK ,MiB                                           *)
(*   Date: 20.11.2012                                        *)
(*   Rev.: 1.1                                               *)
(* ========================================================= *)

HLI3_ChannelSetSingleBlock := FALSE;
IF NOT HLI3_CheckChannelValid(nChannel := nChanIdx) THEN
	RETURN;
END_IF
gpCh[nChanIdx]^.bahn_mc_control.single_block.command_w   := bSingleBlock;

HLI3_ChannelSetSingleBlock := TRUE;

END_FUNCTION

// CNC/3 Control/HLI3_ChannelSetReducedFeed
FUNCTION HLI3_ChannelSetReducedFeed : BOOL
VAR_INPUT
	/// Number of channel 
	nChanIdx: INT;
	bReducedFeed: BOOL;
END_VAR

(* ========================================================= *)
(*    FUN: HLI_ChannelSetReducedFeed                         *)
(* --------------------------------------------------------- *)
(*   Desc:                                                   *)
(* Author: MK,MiB                                            *)
(*   Date: 20.11.2012                                        *)
(*   Rev.: 1.1                                               *)
(* ========================================================= *)


HLI3_ChannelSetReducedFeed := FALSE;
IF NOT HLI3_CheckChannelValid(nChannel := nChanIdx) THEN
	RETURN;
END_IF
gpCh[nChanIdx]^.bahn_mc_control.reduced_speed.command_w := bReducedFeed;
HLI3_ChannelSetReducedFeed := TRUE;

END_FUNCTION

// CNC/3 Control/HLI3_GetChannelStatusInfo
FUNCTION HLI3_GetChannelStatusInfo : BOOL
VAR_INPUT
	/// Number of channel 
	nChanIdx: INT;
END_VAR
VAR
	pChannel: POINTER TO ST_CNCChannel;
END_VAR

(* ========================================================= *)
(*    FUN: HLI_GetStatusInfo                                 *)
(* --------------------------------------------------------- *)
(*   Desc: Status Info from the HLI Interface                *)
(* Author: MK,Mib                                            *)
(*   Date: 18.07.2002                                        *)
(*   Rev.: 1.0                                               *)
(* ========================================================= *)

IF NOT HLI3_CheckChannelValid(nChannel := nChanIdx) THEN
	RETURN;
END_IF


pChannel := ADR(CNCSystem.Channel[nChanIdx]);
pChannel^.ActMode := HLI3_GetChannelMode(nChanIdx:=nChanIdx);
pChannel^.ActState := HLI3_GetChannelState(nChanIdx:=nChanIdx);

pChannel^.Mode.Standby := FALSE;
pChannel^.Mode.Auto := FALSE;
pChannel^.Mode.Homing := FALSE;
pChannel^.Mode.MDI := FALSE;
pChannel^.Mode.Manual := FALSE;

(* Translate mode *)
CASE pChannel^.ActMode OF
	HLI_IMCM_MODE:					pChannel^.ActModeString := 'Mode';
	HLI_IMCM_STANDBY_MODE:			pChannel^.ActModeString := 'StandbyMode'; pChannel^.Mode.Standby:=TRUE;
	HLI_IMCM_AUTOMATIC_MODE:		pChannel^.ActModeString := 'AutomaticMode'; pChannel^.Mode.Auto:=TRUE;
	HLI_IMCM_MDI_MODE:				pChannel^.ActModeString := 'MDIMode'; pChannel^.Mode.MDI:=TRUE;
	HLI_IMCM_MANUAL_MODE:			pChannel^.ActModeString := 'ManualMode'; pChannel^.Mode.Manual:=TRUE;;
	HLI_IMCM_REFERENCE_MODE:		pChannel^.ActModeString := 'ReferenceMode'; pChannel^.Mode.Homing:=TRUE;
ELSE
	pChannel^.ActModeString := '---';
END_CASE;

pChannel^.State.Selected:=FALSE;
pChannel^.State.Ready:=FALSE;
pChannel^.State.Active:=FALSE;
pChannel^.State.Hold:=FALSE;

(* Translate state *)
CASE pChannel^.ActState OF
	HLI_IMCM_PROCESS_DESELECTED:	pChannel^.ActStateString := 'Deselected';
	HLI_IMCM_PROCESS_SELECTED:		pChannel^.ActStateString := 'Selected'; pChannel^.State.Selected:=TRUE;
	HLI_IMCM_PROCESS_READY:			pChannel^.ActStateString := 'Ready'; pChannel^.State.Ready:=TRUE;
	HLI_IMCM_PROCESS_ACTIVE:		pChannel^.ActStateString := 'Active'; pChannel^.State.Active:=TRUE;
	HLI_IMCM_PROCESS_HOLD:			pChannel^.ActStateString := 'Hold'; pChannel^.State.Hold:=TRUE;
	HLI_IMCM_PROCESS_ERROR:			pChannel^.ActStateString := 'Error';
	HLI_IMCM_PROCESS_SELECTING:		pChannel^.ActStateString := 'Selecting';
	HLI_IMCM_PROCESS_DESELECTING:	pChannel^.ActStateString := 'Deselecting';
	HLI_IMCM_PROCESS_PREPARING:		pChannel^.ActStateString := 'Preparing';
	HLI_IMCM_PROCESS_CLEARING:		pChannel^.ActStateString := 'Clearing';
	HLI_IMCM_PROCESS_STARTING:		pChannel^.ActStateString := 'Starting';
	HLI_IMCM_PROCESS_ABORTING:		pChannel^.ActStateString := 'Aborting';
	HLI_IMCM_PROCESS_STOPPING:		pChannel^.ActStateString := 'Stopping';
	HLI_IMCM_PROCESS_RESUMING:		pChannel^.ActStateString := 'Resuming';
	HLI_IMCM_PROCESS_RESETTING:		pChannel^.ActStateString := 'Resetting';
	HLI_IMCM_PROCESS_FINISHING:		pChannel^.ActStateString := 'Finishing';
ELSE
	pChannel^.ActStateString := '---';
END_CASE;

END_FUNCTION

// CNC/3 Control/HLI3_GetChannelMode
FUNCTION HLI3_GetChannelMode : UDINT
VAR_INPUT
	/// Number of channel 
	nChanIdx: INT;
END_VAR

(* ========================================================= *)
(*    FUN: HLI_GetChannelMode                                *)
(* --------------------------------------------------------- *)
(*   Desc:                                                   *)
(* Author: MK                                                *)
(*   Date: 18.07.2002                                        *)
(*   Rev.: 1.0                                               *)
(* ========================================================= *)
HLI3_GetChannelMode := 0;
IF NOT HLI3_CheckChannelValid(nChannel := nChanIdx) THEN
	RETURN;
END_IF

(* if the stop button from the HMI is selected the request is set *)
HLI3_GetChannelMode := gpCh[nChanIdx]^.channel_mc_control.mode_and_state.state_r.mode;

END_FUNCTION

// CNC/3 Control/HLI3_GetChannelState
FUNCTION HLI3_GetChannelState : UDINT
VAR_INPUT
	/// Number of channel 
	nChanIdx: INT;
END_VAR

(* ========================================================= *)
(*    FUN: HLI3_GetChannelState                              *)
(* --------------------------------------------------------- *)
(*   Desc:                                                   *)
(* Author: MK                                                *)
(*   Date: 18.07.2002                                        *)
(*   Rev.: 1.0                                               *)
(* ========================================================= *)

HLI3_GetChannelState := 0;
IF NOT HLI3_CheckChannelValid(nChannel := nChanIdx) THEN
	RETURN;
END_IF

(* if the stop button from the HMI is selected the request is set *)
HLI3_GetChannelState := gpCh[nChanIdx]^.channel_mc_control.mode_and_state.state_r.state;

END_FUNCTION

// CNC/3 Control/HLI3_GetChannelError
FUNCTION HLI3_GetChannelError : BOOL
VAR_INPUT
	/// Number of channel 
	nChanIdx: INT;
END_VAR
VAR
	pChannel: POINTER TO ST_CNCChannel;
END_VAR

(* ========================================================= *)
(*    FUN: HLI_GetChannelError                               *)
(* --------------------------------------------------------- *)
(*   Desc: Gets the channel error                            *)
(* Return: The error flag of the channel                     *)
(* Author: MK , MiB, TV                                      *)
(*   Date: 08.07.2015                                        *)
(*   Rev.: 1.3                                               *)
(* ========================================================= *)

IF NOT HLI3_CheckChannelValid(nChannel := nChanIdx) THEN
	RETURN;
END_IF

pChannel := ADR(CNCSystem.Channel[nChanIdx]);

(* Visualisation of Mode and State *)
pChannel^.ActMode  := HLI3_GetChannelMode(nChanIdx:=nChanIdx);
pChannel^.ActState := HLI3_GetChannelState(nChanIdx:=nChanIdx);

(* Error messages id *)
IF pChannel^.ActState = HLI_IMCM_PROCESS_ERROR THEN
	pChannel^.Error := TRUE;	
ELSE
	pChannel^.Error := FALSE;	
END_IF

END_FUNCTION

// CNC/4 MHT-Function/HLI3_QuitChannelMHTFunction
FUNCTION_BLOCK HLI3_QuitChannelMHTFunction
VAR_INPUT
	/// Number of channel 
	nChanIdx: INT;
	bM30Acknowledgement : BOOL;
END_VAR
VAR_OUTPUT
	bOK: BOOL;
END_VAR
VAR
	ChannelMFunction: HLI3_DoChannelMFunction;
	ChannelTFunction: HLI3_DoChannelTFunction;
	ChannelHFunction: HLI3_DoChannelHFunction;
	/// local pointer to Data of actual Channel 
	pChannelData: POINTER TO HIGH_LEVEL_INTERFACE_CH;
	/// local pointer to actual techno unit 
	pActTechnoUnit: POINTER TO TECHNO_UNIT_CH;
	/// Index of axis specific technology function at HLI 
	nTechFctMaxIdx: UINT;
	nTechFctAnzahl : UINT; 
	/// loop variable 
	idx: UINT;
	/// number of M-function 
	nFuncNr: UDINT;
	nArgument: DINT;
	/// basis id of a tool 
	nToolBasicId: UDINT;
	pMHProcess: POINTER TO HLI_M_H_PROZESS;
	pSProcess: POINTER TO HLI_S_PROZESS;
	pTProcess: POINTER TO HLI_T_PROZESS;
	stAttributeData: St_TechnoAttributeData;	
END_VAR

(* ========================================================= *)
(*     FB: HLI3_QuitChannelMHTFunction                        *)
(* --------------------------------------------------------- *)
(*   Desc:                                                   *)
(* Author: MK                                                *)
(*   Rev.: 1.1                                               *)
(*   Date: 18.07.2002                                        *)
(*       : 08.04.2005                                        *)
(*          24.11.2010 MiB Erweiterung um H Funktionen 		 *)
(* ========================================================= *)
(* Rev.:	1.2												 *)
(* Date:	02.10.2010                                    	 *)
(* Author:	HR												 *)
(* Author:	Added support for additional m function number	 *)
(* ========================================================= *)
(* Rev.:	1.3												 *)
(* Date:	26.01.2011                                    	 *)
(* Author:	HR												 *)
(* Author:	Added support for additional h function number	 *)
(* ========================================================= *)
(* Rev.:	1.4												 *)
(* Date:	20.11.2012                                    	 *)
(* Author:	MiB												 *)
(* Author:	TC3												 *)
(* ========================================================= *)
(* Rev.:	1.4.1									         *)
(* Date:	15.07.2013                                    	 *)
(* Author:	TV												 *)
(* ========================================================= *)
(* Rev.:	1.4.2									         *)
(* Date:	22.09.2016                                    	 *)
(* Author:	TV												 *)
(* ========================================================= *)
(* ========================================================= *)
(* Rev.:	1.4.3									         *)
(* Date:	01.12.2017                                    	 *)
(* Author:	TV												 *)
(*													 	 	 *)
(* ========================================================= *)

IF NOT HLI3_CheckChannelValid(nChannel := nChanIdx) THEN
	bOK := FALSE;
	RETURN; (* A b b r u c h *)
END_IF


(* get pointer to channel data *)
pChannelData := gpCh[nChanIdx];

pActTechnoUnit := ADR(pChannelData^.techno_unit_std_sync[0]);

(* test if there are open synchronisations  *)
IF pChannelData^.used_units_std_sync_r > 0 THEN

	nTechFctAnzahl := pChannelData^.used_units_std_sync_r;
	
	IF nTechFctAnzahl  > 0 THEN

        nTechFctMaxIdx := nTechFctAnzahl  - 1;  

		FOR idx := 0 TO nTechFctMaxIdx DO
			(* get pointer to actual techno unit *)
			pActTechnoUnit := ADR(pChannelData^.techno_unit_std_sync[idx]);
		
		
			(* test if this M-function has to be acknowledged *)
			IF pActTechnoUnit^.please_rw = TRUE AND				(* request from CNC *)
			   pActTechnoUnit^.done_w = FALSE AND				(* not acknowledged *)
			   pActTechnoUnit^.fkt_ctrl_r = HLI_INTF_M_FKT		(* M-function *)
			THEN
				(* Read number of M-function *)
				pMHProcess := ADR(pActTechnoUnit^.attribut_r.data[0]);
				nFuncNr    := pMHProcess^.nr;
				nArgument	:= pMHProcess^.add_nr_r;
				
				
				stAttributeData.nFunctionNumber_r := pMHProcess^.nr;
				stAttributeData.nTime_r		:= pMHProcess^.zeit;
				stAttributeData.nArgument_r 		:= pMHProcess^.add_nr_r;
				stAttributeData.nBlockNumber_r 	:= pMHProcess^.satz_nr;
				stAttributeData.nPrgLineNumber_r	:= pMHProcess^.prg_zeilen_nr;
				
		
				ChannelMFunction(nChanIdx:=nChanIdx, stTechnoAttributeData := stAttributeData, bM30Acknowledgement := bM30Acknowledgement);
				IF ChannelMFunction.bBusy = FALSE THEN
					(* acknowledge this M-function *)
					pActTechnoUnit^.please_rw := FALSE;
					pActTechnoUnit^.done_w := TRUE;				
				END_IF
		
				bOK := TRUE;
			END_IF
	
	
			(* test if this H-function has to be acknowledged *)
			IF pActTechnoUnit^.please_rw = TRUE AND						(* request from CNC *)
			   pActTechnoUnit^.done_w = FALSE AND						(* not acknowledged *)
			   pActTechnoUnit^.fkt_ctrl_r = HLI_INTF_H_FKT		(* H-function *)
			THEN
				(* Read number of H-function *)
				pMHProcess := ADR(pActTechnoUnit^.attribut_r.data[0]);
				stAttributeData.nFunctionNumber_r := pMHProcess^.nr;
				stAttributeData.nTime_r		:= pMHProcess^.zeit;
				stAttributeData.nArgument_r 		:= pMHProcess^.add_nr_r;
				stAttributeData.nBlockNumber_r 	:= pMHProcess^.satz_nr;
				stAttributeData.nPrgLineNumber_r	:= pMHProcess^.prg_zeilen_nr;
		
				ChannelHFunction(nChanIdx:=nChanIdx, stTechnoAttributeData:= stAttributeData);
	
				(* acknowledge this H-function *)
				IF ChannelHFunction.bBusy = FALSE THEN
						(* acknowledge this H-function *)
					pActTechnoUnit^.please_rw := FALSE;
					pActTechnoUnit^.done_w := TRUE;			
				END_IF
				bOK := TRUE;
			END_IF
		
			(* test if this T-function has to be acknowledged *)
			IF pActTechnoUnit^.please_rw = TRUE AND				(* request from CNC *)
			   pActTechnoUnit^.done_w = FALSE AND				(* not acknowledged *)
			   pActTechnoUnit^.fkt_ctrl_r = HLI_INTF_TOOL		(* T-function *)
			THEN
				(* Read number of T-function *)
				pTProcess    := ADR(pActTechnoUnit^.attribut_r.data[0]);
				nToolBasicId := DINT_TO_UDINT(pTProcess^.id.basic);
		
				ChannelTFunction(nChanIdx:=nChanIdx, nFuncNr:=nToolBasicId);
		
				(* acknowledge this T-function *)
				pActTechnoUnit^.please_rw := FALSE;
				pActTechnoUnit^.done_w := TRUE;				
				bOK := TRUE;
			END_IF
		
		END_FOR
	
	END_IF

END_IF


(*
	HLI_INTF_H_FKT                 :    INT:=2;
	HLI_INTF_SPINDEL              :    INT:=3;
	HLI_INTF_TOOL                 :    INT:=4;
	GCW_250_HLIIntfAxBlock              :    INT:=5;
	GCW_250_HLIIntfVEVariable           :    INT:=6;
	GCW_250_HLIIntfVEVariable_1         :    INT:=7;
	GCW_250_HLIIntfVEVariable_2         :    INT:=8;
	GCW_250_HLIIntfUnknown              :    INT:=9;
*)

(*******************************************************************************************************************)

FOR idx := 0 TO INT_TO_UINT(HLI_TU_CH_LATE_SYNC_MAXIDX) DO
	IF pChannelData^.techno_unit_late_sync[idx].please_rw = TRUE
	AND pChannelData^.techno_unit_late_sync[idx].done_w = FALSE THEN

		(* get pointer to actual techno unit *)
		pActTechnoUnit := ADR(pChannelData^.techno_unit_late_sync[idx]);

		IF pActTechnoUnit^.please_rw = TRUE AND				(* request from CNC *)
			pActTechnoUnit^.done_w = FALSE AND				(* not acknowledged *)
			pActTechnoUnit^.fkt_ctrl_r = HLI_INTF_M_FKT		(* M-function *)
		THEN
			pMHProcess := ADR(pActTechnoUnit^.attribut_r.data[0]);
			nFuncNr    := pMHProcess^.nr;
			
			stAttributeData.nFunctionNumber_r := pMHProcess^.nr;
			stAttributeData.nTime_r		:= pMHProcess^.zeit;
			stAttributeData.nArgument_r 		:= pMHProcess^.add_nr_r;
			stAttributeData.nBlockNumber_r 	:= pMHProcess^.satz_nr;
			stAttributeData.nPrgLineNumber_r	:= pMHProcess^.prg_zeilen_nr;

			ChannelMFunction(nChanIdx:=nChanIdx, stTechnoAttributeData:=stAttributeData);
			IF ChannelMFunction.bBusy = FALSE THEN
			(* acknowledge this M-function *)
			pActTechnoUnit^.please_rw := FALSE;
			pActTechnoUnit^.done_w := TRUE;
			
			(* ADSLOGDINT( msgCtrlMask := ADSLOG_MSGTYPE_MSGBOX OR
										ADSLOG_MSGTYPE_LOG,
						msgFmtStr := 'Channel acknowledge of M-function: %d',
						dintArg := pMHProcess^.nr);
			*)
		END_IF
		bOK := TRUE;

	(*	ELSIF   pActTechnoUnit^.fkt_ctrl_r = HLI_INTF_SPINDEL THEN (* spindle-function *)

 			(* Example: read number of S-function *)
			pSProzess := ADR(pActTechnoUnit^.attribut_r.data[0]);
			ADSLOGDINT( msgCtrlMask := ADSLOG_MSGTYPE_MSGBOX OR
										ADSLOG_MSGTYPE_LOG,
						msgFmtStr := 'Late synch : %d',
						dintArg := pSProzess^.move_cmd);

		ELSIF   pActTechnoUnit^.fkt_ctrl_r = HLI_INTF_TOOL THEN

			pHLI_T_PROZESS := ADR(pActTechnoUnit^.attribut_r.data[0]);
			ADSLOGDINT( msgCtrlMask := ADSLOG_MSGTYPE_MSGBOX OR
										ADSLOG_MSGTYPE_LOG,
						msgFmtStr := 'Late tool process: %d',
						dintArg := pTProcess^.id.basic);*)
		(*ELSE
				ADSLOGDINT( msgCtrlMask := ADSLOG_MSGTYPE_MSGBOX OR
											ADSLOG_MSGTYPE_LOG,
							msgFmtStr := 'Channel acknowledge unknown type: %d',
							dintArg := pActTechnoUnit^.fkt_ctrl_r);*)
		END_IF

	END_IF
END_FOR
(**********************************************************************************************************************)

END_FUNCTION_BLOCK

// CNC/4 MHT-Function/HLI3_DoChannelMFunction
FUNCTION_BLOCK HLI3_DoChannelMFunction
VAR_INPUT
	/// Channel number 
	nChanIdx: INT;
	stTechnoAttributeData: St_TechnoAttributeData;
	bM30Acknowledgement : BOOL;
END_VAR
VAR_OUTPUT
	bBusy: BOOL;
END_VAR
VAR
	pChannel: POINTER TO ST_CncChannel;
END_VAR

(* ========================================================= *)
(*     FB: HLI_DoChannelMFunction                            *)
(* --------------------------------------------------------- *)
(*   Desc:                                                   *)
(* Author: MK                                                *)
(*   Rev.: 1.1                                               *)
(*   Date: 18.07.2002                                        *)
(*       : 08.04.2005                                        *)
(* ========================================================= *)
(* Rev.:	1.2												 *)
(* Date:	02.10.2010                                   	 *)
(* Author:	HR												 *)
(* Author:	Added support for additional m function number	 *)
(*			via new input variable 'nArg'				 	 *)
(* ========================================================= *)
(* Rev.:	1.3												 *)
(* Date:	23.11.2012                                   	 *)
(* Author:	TV, MiB											 *)
(* Author:	structure St_TechnoAttributeData instead of      *)
(*			simple bool array	 							 *)
(* ========================================================= *)
(* Rev.:	1.4												 *)
(* Date:	22.09.2016                                   	 *)
(* Author:	TV 											 	 *)
(* Dec:		Implementation of Input bM30Acknowledgement      *)
(*				 							                 *)
(* ========================================================= *)

bBusy := TRUE;
IF NOT HLI3_CheckChannelValid(nChannel := nChanIdx) THEN
	RETURN; (* A b b r u c h *)
END_IF


pChannel := ADR(CNCSystem.Channel[nChanIdx]);

(* Synch M-Functions *)
IF stTechnoAttributeData.nFunctionNumber_r > 0 AND stTechnoAttributeData.nFunctionNumber_r < 1000 THEN
	IF NOT pChannel^.M[stTechnoAttributeData.nFunctionNumber_r].bRes THEN					(* M-Function not set *)
		pChannel^.M[stTechnoAttributeData.nFunctionNumber_r].bState_rw				:= TRUE;	(* set M-Function *)
		pChannel^.M[stTechnoAttributeData.nFunctionNumber_r].nArgument_r		:= stTechnoAttributeData.nArgument_r;
		pChannel^.M[stTechnoAttributeData.nFunctionNumber_r].nBlockNumber_r		:= stTechnoAttributeData.nBlockNumber_r;
		pChannel^.M[stTechnoAttributeData.nFunctionNumber_r].nPrgLineNumber_r	:= stTechnoAttributeData.nPrgLineNumber_r;
		pChannel^.M[stTechnoAttributeData.nFunctionNumber_r].nFunctionNumber_r	:= stTechnoAttributeData.nFunctionNumber_r;
		pChannel^.M[stTechnoAttributeData.nFunctionNumber_r].nTime_r			:= stTechnoAttributeData.nTime_r;		
		pChannel^.M[stTechnoAttributeData.nFunctionNumber_r].bRes 				:= TRUE;	(* set acknowledge *)
		pChannel^.actM_r := CONCAT('M', UDINT_TO_STRING(stTechnoAttributeData.nFunctionNumber_r));
	ELSE
		IF NOT pChannel^.M[stTechnoAttributeData.nFunctionNumber_r].bState_rw THEN				(* wait for quit *)
			pChannel^.M[stTechnoAttributeData.nFunctionNumber_r].bRes 			:= FALSE;	(* quit the ack *)
			pChannel^.M[stTechnoAttributeData.nFunctionNumber_r].nArgument_r	:= 0;		(* reset the argument *)
			pChannel^.M[stTechnoAttributeData.nFunctionNumber_r].nBlockNumber_r		:= 0;
			pChannel^.M[stTechnoAttributeData.nFunctionNumber_r].nPrgLineNumber_r	:= 0;
			pChannel^.M[stTechnoAttributeData.nFunctionNumber_r].nFunctionNumber_r	:= 0;
			pChannel^.M[stTechnoAttributeData.nFunctionNumber_r].nTime_r			:= 0;				
			pChannel^.actM_r :='';
			bBusy 							:= FALSE;	(* quit *)
		END_IF
	END_IF
END_IF


(* Quit M00, M01, M02 , M17, M29, M30 *)
IF 	stTechnoAttributeData.nFunctionNumber_r = 0 OR 
	stTechnoAttributeData.nFunctionNumber_r = 01 OR 
	stTechnoAttributeData.nFunctionNumber_r = 02 OR 
	stTechnoAttributeData.nFunctionNumber_r = 17  OR 
	stTechnoAttributeData.nFunctionNumber_r = 29  OR 
	(stTechnoAttributeData.nFunctionNumber_r = 30 AND bM30Acknowledgement) THEN
		pChannel^.M[stTechnoAttributeData.nFunctionNumber_r].bState_rw 			:= FALSE;
		pChannel^.M[stTechnoAttributeData.nFunctionNumber_r].nArgument_r	:= 0;
		pChannel^.M[stTechnoAttributeData.nFunctionNumber_r].bRes 			:= FALSE;
		bBusy 							:= FALSE;
END_IF

END_FUNCTION_BLOCK

// CNC/4 MHT-Function/HLI3_DoChannelTFunction
FUNCTION_BLOCK HLI3_DoChannelTFunction
VAR_INPUT
	/// Channel number 
	nChanIdx: INT;
	/// Number of T-function 
	nFuncNr: UDINT;
END_VAR
VAR_OUTPUT
	bBusy: BOOL;
END_VAR
VAR
	bStartTimer: BOOL;
END_VAR

(* ========================================================= *)
(*     FB: HLI_DoChannelTFunction                            *)
(* --------------------------------------------------------- *)
(*   Desc:                                                   *)
(* Author: MK, MiB                                           *)
(*   Rev.: 1.1                                               *)
(*   Date: 18.07.2002                                        *)
(*       : 08.04.2005, 03.03.2016 							 *)
(* ========================================================= *)


bBusy := FALSE;
RETURN;

IF NOT HLI3_CheckChannelValid(nChannel := nChanIdx) THEN
	RETURN; (* A b b r u c h *)
END_IF
bBusy := TRUE;

CASE nChanIdx OF
	0:	(* cnc channel 1 -------------------------------------- *)
		CASE nFuncNr OF
			0:		bBusy := FALSE;
			1:		bBusy := FALSE;
			2:		bBusy := FALSE;
			3:		bBusy := FALSE;
			4:		bBusy := FALSE;
			5:		bBusy := FALSE;
			6:		bBusy := FALSE;
			7:		bBusy := FALSE;
			8:		bBusy := FALSE;

			ELSE
			ADSLOGDINT( msgCtrlMask :=    ADSLOG_MSGTYPE_MSGBOX
			                           OR ADSLOG_MSGTYPE_LOG,
						msgFmtStr   := 'T-Funktion (%d), Channel 1, HLI_DoChannelTFunction() not implemented!',
						dintArg     := UDINT_TO_DINT(nFuncNr));
				(* Quit the M-Function *)
				bBusy := TRUE;
		END_CASE;


	1:	(* cnc channel 2 -------------------------------------- *)
		CASE nFuncNr OF
			0:		bBusy := FALSE;
			1:		bBusy := FALSE;
			2:		bBusy := FALSE;
			3:		bBusy := FALSE;


			ELSE
				ADSLOGDINT( msgCtrlMask :=    ADSLOG_MSGTYPE_MSGBOX
				                           OR ADSLOG_MSGTYPE_LOG,
							msgFmtStr   := 'T-Funktion (%d), Channel 2, HLI_DoChannelTFunction() not implemented!',
							dintArg     := UDINT_TO_DINT(nFuncNr));
				(* Quit the M-Function *)
				bBusy := FALSE;
		END_CASE;

ELSE
	ADSLOGDINT( msgCtrlMask :=    ADSLOG_MSGTYPE_MSGBOX
	                           OR ADSLOG_MSGTYPE_LOG,
				msgFmtStr   := 'Unknown channel number (%d) in HLI_DoChannelTFunction',
				dintArg     := INT_TO_DINT(nChanIdx));
	bBusy := FALSE;
END_CASE;

END_FUNCTION_BLOCK

// CNC/4 MHT-Function/HLI3_DoChannelHFunction
FUNCTION_BLOCK HLI3_DoChannelHFunction
VAR_INPUT
	/// Channel number 
	nChanIdx: INT;
	stTechnoAttributeData: St_TechnoAttributeData;
END_VAR
VAR_OUTPUT
	bBusy: BOOL;
END_VAR
VAR
	pChannel: POINTER TO ST_CncChannel;
END_VAR

(* ========================================================= *)
(*     FB: HLI_DoChannelHFunction                            *)
(* --------------------------------------------------------- *)
(*   Desc:                                                   *)
(* Author: MiB                                               *)
(*   Rev.: 1.0                                               *)
(*   Date: 24.11.2010                                        *)
(*       : 08.04.2005                                        *)
(* ========================================================= *)
(* Rev.:	1.2												 *)
(* Date:	26.01.2011                                   	 *)
(* Author:	HR												 *)
(* Author:	Added support for additional h function number	 *)
(*			via new input variable 'nArg'				 	 *)
(* ========================================================= *)
bBusy := TRUE;

IF NOT HLI3_CheckChannelValid(nChannel := nChanIdx) THEN
	RETURN; (* A b b r u c h *)
END_IF


pChannel := ADR(CNCSystem.Channel[nChanIdx]);

(* Synch M-Functions *)
IF stTechnoAttributeData.nFunctionNumber_r > 0 AND stTechnoAttributeData.nFunctionNumber_r < 1000 THEN
	IF NOT pChannel^.H[stTechnoAttributeData.nFunctionNumber_r].bRes THEN					(* M-Function not set *)
		pChannel^.H[stTechnoAttributeData.nFunctionNumber_r].bState_rw				:= TRUE;	(* set M-Function *)
		pChannel^.H[stTechnoAttributeData.nFunctionNumber_r].nArgument_r		:= stTechnoAttributeData.nArgument_r;
		pChannel^.H[stTechnoAttributeData.nFunctionNumber_r].nBlockNumber_r		:= stTechnoAttributeData.nBlockNumber_r;
		pChannel^.H[stTechnoAttributeData.nFunctionNumber_r].nPrgLineNumber_r	:= stTechnoAttributeData.nPrgLineNumber_r;
		pChannel^.H[stTechnoAttributeData.nFunctionNumber_r].nFunctionNumber_r	:= stTechnoAttributeData.nFunctionNumber_r;
		pChannel^.H[stTechnoAttributeData.nFunctionNumber_r].nTime_r			:= stTechnoAttributeData.nTime_r;		
		pChannel^.H[stTechnoAttributeData.nFunctionNumber_r].bRes 				:= TRUE;	(* set acknowledge *)
		pChannel^.actH_r := CONCAT('H', UDINT_TO_STRING(stTechnoAttributeData.nFunctionNumber_r));
	ELSE
		IF NOT pChannel^.H[stTechnoAttributeData.nFunctionNumber_r].bState_rw THEN				(* wait for quit *)
			pChannel^.H[stTechnoAttributeData.nFunctionNumber_r].bRes 			:= FALSE;	(* quit the ack *)
			pChannel^.H[stTechnoAttributeData.nFunctionNumber_r].nArgument_r	:= 0;		(* reset the argument *)
			pChannel^.H[stTechnoAttributeData.nFunctionNumber_r].nBlockNumber_r		:= 0;
			pChannel^.H[stTechnoAttributeData.nFunctionNumber_r].nPrgLineNumber_r	:= 0;
			pChannel^.H[stTechnoAttributeData.nFunctionNumber_r].nFunctionNumber_r	:= 0;
			pChannel^.h[stTechnoAttributeData.nFunctionNumber_r].nTime_r			:= 0;
			pChannel^.actH_r := '';					
			bBusy 							:= FALSE;	(* quit *)
		END_IF
	END_IF
END_IF

END_FUNCTION_BLOCK

// CNC/3 Control/FB_Diag
FUNCTION_BLOCK FB_Diag
VAR_OUTPUT
	Alarm: BOOL;
	Vorwarn: BOOL;
	Meld: BOOL;
END_VAR

Alarm := TRUE;
Vorwarn := TRUE;
Meld := TRUE;

END_FUNCTION_BLOCK

// CNC/3 Control/HLI3_ChannelSetSuspendAxisOutput
FUNCTION HLI3_ChannelSetSuspendAxisOutput : BOOL
VAR_INPUT
	/// Number of channel 
	nChanIdx: INT;
	bSuspendAxis: BOOL;
END_VAR

(* ========================================================= *)
(*    FUN: HLI_ChannelSuspendAxisOutput                      *)
(* --------------------------------------------------------- *)
(*   Desc:                                                   *)
(* Author: MK , MiB                                          *)
(*   Date: 20.11.2012                                        *)
(*   Rev.: 1.1                                               *)
(* ========================================================= *)
HLI3_ChannelSetSuspendAxisOutput := TRUE;
IF NOT HLI3_CheckChannelValid(nChannel := nChanIdx) THEN
	RETURN;
END_IF
gpCh[nChanIdx]^.bahn_mc_control.suspend_axis_output.command_w := bSuspendAxis;
HLI3_ChannelSetSuspendAxisOutput := TRUE;

END_FUNCTION

// CNC/3 Control/HLI3_GetActualAxisPos
FUNCTION HLI3_GetActualAxisPos : LREAL
VAR_INPUT
	///Achs ID
	nHliAxisIdx: INT;
END_VAR
VAR
	HLI_GetActualAxisPos: DINT;
END_VAR



IF NOT (HLI3_CheckAxisValid(nHliAxisIdx := nHliAxisIdx)) THEN
	HLI3_GetActualAxisPos := -1;
	RETURN;
END_IF

HLI3_GetActualAxisPos:=  gpAx[nHliAxisIdx]^.lr_state.current_position_acs_r;

END_FUNCTION

// CNC/3 Control/HLI3_GetAxisReferenceState
FUNCTION HLI3_GetAxisReferenceState : BOOL
VAR_INPUT
	nHliAxisIdx: INT;
END_VAR


IF NOT HLI3_CheckAxisValid(nHliAxisIdx := nHliAxisIdx) THEN
	HLI3_GetAxisReferenceState := FALSE;
	RETURN;
END_IF

HLI3_GetAxisReferenceState:= gpAx[nHliAxisIdx]^.lr_state.homing_done_r;

END_FUNCTION

// CNC/3 Control/HLI3_GetChannelActiveG
FUNCTION_BLOCK HLI3_GetChannelActiveG
VAR_INPUT
	bExec:	   BOOL;			// riding edge to start read
	nChanIdx: INT;    			// zero based channel index	
END_VAR
VAR_OUTPUT
	ActiveG : ARRAY[0..39] OF INT;
	bBusy: BOOL;
	bError: BOOL;
	nErrorID: UDINT;
END_VAR
VAR
	fbAdsRead: ADSREAD;
END_VAR

(* ========================================================= *)
(*    FUN: HLI3_GetChannelActiveG                   		 *)
(* --------------------------------------------------------- *)
(*   Desc: Gets the channel specific active G functions      *)
(*															 *)
(* Return: Array[0..39] filled with the G information (<> -1)*)
(* Author: MiB                                               *)
(*   Date: 12.01.2016                                        *)
(*   Rev.: 1.0                                               *)
(* ========================================================= *)

fbAdsRead(
	NETID:= '' , 
	PORT:= 553, 
	IDXGRP:= 16#20100 + INT_TO_UDINT(nChanIdx) + 1, 
	IDXOFFS:= 16#3C , 
	LEN:= SIZEOF(ActiveG) , 
	DESTADDR:= ADR(ActiveG),
	READ:= bExec, 
	TMOUT:= , 
	BUSY=> bBusy, 
	ERR=> bError, 
	ERRID=> nErrorId );

END_FUNCTION_BLOCK

// CNC/3 Control/HLI3_GetChannelMessage
FUNCTION_BLOCK HLI3_GetChannelMessage
VAR_INPUT
	/// Number of channel 
	nChanIdx: INT;
	bExecute: BOOL := FALSE;
	bShowDlg: BOOL := FALSE;
END_VAR
VAR_OUTPUT
	strToPLC: STRING(HLI_MSG_CONTENT_STRL) := '';
	iMsgType: DWORD := 0;
END_VAR
VAR
	pChannel: POINTER TO HIGH_LEVEL_INTERFACE_CH;
	pMsgCU: POINTER TO MC_CONTROL_MSG_UNIT;
	pMsgToPLC: POINTER TO STRING(HLI_MSG_CONTENT_STRL);
END_VAR

(* ========================================================= *)
(*     FB: HLI_GetChannelMessage                             *)
(* --------------------------------------------------------- *)
(*   Desc: Get message from the CNC                          *)
(*   Author: MK, MiB                                         *)
(*   Date: 20.11.2012                                        *)
(*   Last:                                                   *)
(*   Rev.: 1.01                                              *)
(* ========================================================= *)

IF NOT HLI3_CheckChannelValid(nChannel := nChanIdx) THEN
	RETURN;
END_IF


(* Get pointer to data of a specific channel at the HLI *)
pChannel := gpCh[nChanIdx];

(* Control unit at the HLI that handles channel specific messages *)
pMsgCU := ADR(pChannel^.msg_mc_control);

IF bExecute = TRUE THEN
	(* Is the complete message in the control unit? *)
	IF pMsgCU^.request_semaphor_rw = TRUE
	THEN
		(* Pointer to content of the message sent to the PLC *)
		pMsgToPLC := ADR(pMsgCU^.request_r.inhalt);

		(* Get the message from the control unit *)
		strToPLC := pMsgToPLC^;

   	    CNCSystem.Channel[nChanIdx].Message := strToPLC;

		(* Get the message type *)
		iMsgType := pMsgCU^.request_r.typ;

		(* Pop up dialog with the message send to the PLC *)
		IF bShowDlg THEN
			ADSLOGSTR( msgCtrlMask := ADSLOG_MSGTYPE_MSGBOX OR ADSLOG_MSGTYPE_LOG,
			           msgFmtStr   := 'Message sent to PLC via HLI:%s',
			           strArg      := strToPLC);
		END_IF

		(* Acknowledge that you got the message *)
		pChannel^.msg_mc_control.request_semaphor_rw  := FALSE;
	END_IF;
END_IF;

END_FUNCTION_BLOCK

// CNC/3 Control/HLI3_GetFeedholdState
FUNCTION HLI3_GetFeedholdState : BOOL
VAR_INPUT
	/// Number of channel 
	nChanIdx: INT;
END_VAR


IF NOT HLI3_CheckChannelValid(nChannel := nChanIdx) THEN
	RETURN;
END_IF
HLI3_GetFeedholdState:=gpCh[nChanIdx]^.bahn_mc_control.feedhold.state_r;

END_FUNCTION

// CNC/3 Control/HLI3_GetIpoState
FUNCTION HLI3_GetIpoState : BOOL
VAR_INPUT
	nChanIdx: INT;
END_VAR



IF NOT HLI3_CheckChannelValid(nChannel := nChanIdx) THEN
	RETURN;
END_IF

HLI3_GetIpoState:=gpCh[nChanIdx]^.bahn_state.interpolation_active_r;

END_FUNCTION

// CNC/3 Control/HLI3_HandleSpindleTechno
FUNCTION_BLOCK HLI3_HandleSpindleTechno
VAR_INPUT
	/// Logical axis number of the plc spindle 
	nHliAxisIdx: INT;
	/// The channel which commands the spindle, only used if 'bIsChannelSpecific' set TRUE 
	nHliChannelIdx: INT;
	/// Has to be set TRUE if the spindel intechno function is transmitted via the channel specific section of the HLI
	bIsChannelSpecific: BOOL;
	/// if using a plc controlled spindle: configured log_ax_nr in channel list 
	nLogAxisNoChannelSpecific: INT;
	/// Has to be set TRUE if zthis FB should car about gear change M functions M40 - M45
	bHandleGearChange: BOOL;
	/// Resets all internal states and variables of this function block 
	bChannelReset: BOOL;
END_VAR
VAR_OUTPUT
	/// Returns the commanded revolution programmed with a M03 or M05 [] 
	nRevolution: DINT;
	/// Returns the target position programmed with a M19 [0.1µm] or [] 
	nPosition: DINT;
	/// Error flag 
	bError: BOOL;
	/// Error id 
	nErrorId: UDINT;
END_VAR
VAR_IN_OUT
	/// Raises if the cnc program encounters a M03 for the relevant spindle. Reset this for acknowledge 
	M03: BOOL;
	/// Raises if the cnc program encounters a M04 for the relevant spindle. Reset this for acknowledge 
	M04: BOOL;
	/// Raises if the cnc program encounters a M05 for the relevant spindle. Reset this for acknowledge 
	M05: BOOL;
	/// Raises if the cnc program encounters a M19 for the relevant spindle. Reset this for acknowledge 
	M19: BOOL;
END_VAR
VAR
	/// Raises if the cnc program encounters a M40 for the relevant spindle. Reset this for acknowledge 
	pM40: POINTER TO BOOL;
	/// Raises if the cnc program encounters a M41 for the relevant spindle. Reset this for acknowledge 
	pM41: POINTER TO BOOL;
	/// Raises if the cnc program encounters a M42 for the relevant spindle. Reset this for acknowledge 
	pM42: POINTER TO BOOL;
	/// Raises if the cnc program encounters a M43 for the relevant spindle. Reset this for acknowledge 
	pM43: POINTER TO BOOL;
	/// Raises if the cnc program encounters a M44 for the relevant spindle. Reset this for acknowledge 
	pM44: POINTER TO BOOL;
	/// Raises if the cnc program encounters a M45 for the relevant spindle. Reset this for acknowledge 
	pM45: POINTER TO BOOL;	


	/// Number of open technology functions 
	nOpenTechnoCount: UINT;
	nOpenTechnoCountLate: UINT;
	
	/// Internal acknowledge signal 
	bAcknowledge: BOOL;
	/// Internal state of M03 request 
	M03_Internal: BOOL;
	/// Internal state of M04 request 
	M04_Internal: BOOL;
	/// Internal state of M05 request 
	M05_Internal: BOOL;
	/// Internal state of M19 request 
	M19_Internal: BOOL;
	/// Internal state of M19 request 
	M40_Internal: BOOL;
	/// Internal state of M19 request 
	M41_Internal: BOOL;
	/// Internal state of M19 request 
	M42_Internal: BOOL;
	/// Internal state of M19 request 
	M43_Internal: BOOL;
	/// Internal state of M19 request 
	M44_Internal: BOOL;
	/// Internal state of M19 request 
	M45_Internal: BOOL;
	/// Index of axis specific HLI area 
	nHliAxIfcIdx: UDINT;
	/// Index of axis specific technology function at HLI 
	nTechFctMaxIdx: UINT;
	nTechFctMaxIdxLate: UINT;
	/// Counting variable for loop processing 
	nLoop: UINT;
	
	/// Pointer to spindle specific data 
	pSProcess: POINTER TO HLI_S_PROZESS;
	pMProcess: POINTER TO HLI_M_H_PROZESS;
	/// Rising trigger of input 'bChannelReset' 
	fbRtrigChannelReset: R_TRIG;
	
	bFirstRun : BOOL := TRUE;
	dummyM40: BOOL;
	dummyM41: BOOL;
	dummyM42: BOOL;
	dummyM43: BOOL;
	dummyM44: BOOL;
	dummyM45: BOOL;
	
END_VAR

(****************************************************************************************)
(* POU:		HLI3_HandlePlcSpindle                      									*)
(* Type:	Function Block																*)
(* Author: 	HR, MiB, TV																    *)
(* Date: 	10/11/10																	*)
(* Rev.: 	1.0																			*)
(* Rev.: 	1.6	14/10/23    															*)
(* ------------------------------------------------------------------------------------ *)
(* Desc:	Function block for handling technology functions of PLC spindles. It works	*)
(*			properly if there is a ation axis in the configuration. The logical 		*)
(*			axis no. 'n' of that axis is used to indetify that spindle in this function	*)
(*			block. This implies a spindle configuration like the folowing:				*)
(*				spdl_anzahl                         1	(maybe more?)					*)
(*				main_spindle_ax_nr                  n	(enter right value there)		*)
(*				main_spindle_name                   S									*)
(*				spindle_m_fct_free                  0									*)
(*				spindel[0].bezeichnung              S1									*)
(*				spindel[0].log_achs_nr              n	(enter right value there)		*)
(*				spindel[0].plc_control              1									*)
(*																						*)
(*			The function block may raise some errors specified by an error id:			*)
(*				+ 10000: axis number not valid!											*)
(*																						*)
(****************************************************************************************)
(* Date:	13/09/16																	*)
(* Author:	RCH																			*)
(* Rev:		1.1																			*)
(* ------------------------------------------------------------------------------------ *)
(* Desc 	Renamed, according to Tc2 version. This FB also works for CNC spindles with	*) 
(*			S or M functions set to inform PLC. 										*)
(****************************************************************************************)
(* Date:	13/09/16																	*)
(* Author:	RCH																			*)
(* Rev:		1.2																			*)
(* ------------------------------------------------------------------------------------ *)
(* Desc 	Introduced new input parameters 'bIsChannelSpecific' and 'nChannelNo' in 	*)
(*			order to make this FB work for PLC spindles which are sending synch.		*)
(*			requests via the channel specific section of the HLI. Here the spindle		*)
(* 			specific parameters have to be set as follows:								*)
(*				spindel[n].plc_control            1			(P-CHAN-00069)				*)
(*				spindel[n].log_achs_nr            m			(P-CHAN-00036)				*)
(*																						*)
(*			The logical axis number in P-CHAN-00036 used for such a spindle must not be	*)
(*			lower than one and must not be used by any other axis. This FB works if the	*)
(*			value of this logical axis number fits the parameter 'nHliAxisIdx' only!	*)
(* 																						*)
(*			In order to guarantee save HLI access the following new error codes have	*)
(*			been introduced:															*)
(*				+ 20000: Channel no lower than one!										*)
(*				+ 20001: Channel number exceeds number of configured channels.			*)
(*				+ 20002: No HLI data for channel.										*)
(****************************************************************************************)
(* Date:	14/01/22																	*)
(* Author:	TV																			*)
(* Rev:		1.3																			*)
(* ------------------------------------------------------------------------------------ *)
(* Desc:	bugfix in function to check nHLIAxisIdx and LogAxisId						*) 
(****************************************************************************************)
(* Date:	14/09/10																	*)
(* Author:	RCH																			*)
(* Rev:		1.4																			*)
(* ------------------------------------------------------------------------------------ *)
(* Desc 	Added optional handling of spindle gear change M functions M40 - M45.		*)
(****************************************************************************************)
(* Date:	14/09/12																	*)
(* Author:	RCH																			*)
(* Rev:		1.5																			*)
(* ------------------------------------------------------------------------------------ *)
(* Desc 	Fixed bug with spindle M functions send by the channel spec. section of the	*)
(*			HLI. So far the channel specific section was used for determining the value *)
(*			of  'nTechFctMaxidx'.														*)
(****************************************************************************************)
(* Date:	14/10/23																	*)
(* Author:	MiB																			*)
(* Rev:		1.6																			*)
(* ------------------------------------------------------------------------------------ *)
(* Desc 	Introduced parameter "nLogAxisNoChannelSpecific" which allows to use a plc  *)
(*			spindle without a simulation axis for the spindle. 				 			*)
(*			This paramater is only used if "bIsChannelSpecific == true"					*)
(*																						*)
(*				spindel[n].plc_control            1			(P-CHAN-00069)				*)
(*				spindel[n].log_achs_nr            m			(P-CHAN-00036)				*)
(*																						*)
(*			The logical axis number in P-CHAN-00036 used for such a spindle must not be	*)
(*			lower than one and must not be used by any other axis. This FB works if the	*)
(*			value of this logical axis number fits the parameter 						*)
(*			'nLogAxisNoChannelSpecific' only!											*)
(****************************************************************************************)
(* Date:	15/03/05																	*)
(* Author:	MiB																			*)
(* Rev:		1.7																			*)
(* ------------------------------------------------------------------------------------ *)
(* Desc 	Removed gearchange m functions from var_in_out							    *)
(*			Created new FB HLI3_SpindleTechnoGearchange									*)
(****************************************************************************************)
(*								Init Pointer to pM40..pM45								*)
(****************************************************************************************)
(* Date:	17/02/03																	*)
(* Author:	MiB																			*)
(* Rev:		1.7																			*)
(* ------------------------------------------------------------------------------------ *)
(* Desc 	Handling of late sync M functions. 											*)
(*			Usage of different structure TECHNO_UNIT_AX and TECHNO_UNIT_CH, depending 	*)
(*			on channel or axis specific specific interface 							 	*)
(****************************************************************************************)



IF bFirstRun THEN
	bFirstRun := FALSE;
	pM40 := ADR(dummyM40);
	pM41 := ADR(dummyM41);
	pM42 := ADR(dummyM42);
	pM43 := ADR(dummyM43);
	pM44 := ADR(dummyM44);
	pM45 := ADR(dummyM45);	
END_IF

A_HandleTechno();

ACTION A_HandleTechno:

(****************************************************************************************)
(*								Cyclic reset of  error flag 							*)
(****************************************************************************************)
bError										:= FALSE;
nErrorId									:= 0;

(****************************************************************************************)
(*							  Check for valid logical axis no.							*)
(****************************************************************************************)
IF NOT bIsChannelSpecific AND NOT HLI3_CheckAxisValid(nHliAxisIdx := nHliAxisIdx) THEN
	bError									:= TRUE;
	nErrorId								:= 10000;
	RETURN;
END_IF

IF NOT HLI3_CheckChannelValid(nChannel := nHliChannelIdx) THEN
	bError									:= TRUE;
	nErrorId								:= 20000;
	RETURN;	
END_IF

(****************************************************************************************)
(*											Reset										*)
(****************************************************************************************)
fbRtrigChannelReset
	(CLK := bChannelReset);

IF fbRtrigChannelReset.Q THEN
	nRevolution		:= 0;
	nPosition		:= 0;
	bAcknowledge	:= FALSE;
	M03				:= FALSE;
	M03_Internal	:= FALSE;
	M04				:= FALSE;
	M04_Internal	:= FALSE;
	M05				:= FALSE;
	M05_Internal	:= FALSE;
	M19				:= FALSE;
	M19_Internal	:= FALSE;	
	pM40^			:= FALSE;
	M40_Internal	:= FALSE;
	pM41^			:= FALSE;
	M41_Internal	:= FALSE;
	pM42^			:= FALSE;
	M42_Internal	:= FALSE;
	pM43^			:= FALSE;
	M43_Internal	:= FALSE;
	pM44^			:= FALSE;
	M44_Internal	:= FALSE;
	pM45^			:= FALSE;
	M45_Internal	:= FALSE;
END_IF

(****************************************************************************************)
(*									Receive requests from cnc							*)
(****************************************************************************************)
(* Look out for open technology function either on the channel or the axis specific		*)
(* section of the HLI, depending on parameter ''.										*)
IF bIsChannelSpecific THEN
	nOpenTechnoCount	:= gpCh[nHliChannelIdx]^.used_units_std_sync_r;
	nOpenTechnoCountLate:= gpCh[nHliChannelIdx]^.used_units_late_sync_r;
	
	nTechFctMaxidx 		:= gpCh[nHliChannelIdx]^.used_units_std_sync_r - 1;
	nTechFctMaxIdxLate 	:= gpCh[nHliChannelIdx]^.used_units_late_sync_r - 1;
ELSE
	nOpenTechnoCount	:= gpAx[nHliAxisIdx]^.used_units_std_sync_r;
	nOpenTechnoCountLate:= gpAx[nHliAxisIdx]^.used_units_late_sync_r;

	nTechFctMaxidx 		:= gpAx[nHliAxisIdx]^.used_units_std_sync_r - 1;
	nTechFctMaxIdxLate 	:= gpAx[nHliAxisIdx]^.used_units_late_sync_r - 1;		
END_IF

IF nOpenTechnoCount > 0 THEN
	FOR nLoop := 0 TO nTechFctMaxIdx DO
		(* Depending on the source determined by parameter 'bIsChannelSpecific', the		*)
		(* channel or axis specific section of the HLI will be examined.					*)
		IF bIsChannelSpecific THEN		
				
			M_HandleTechnoCh(ADR(gpCh[nHliChannelIdx]^.techno_unit_std_sync[nLoop]), M03 := M03, M04 := M04, M05 := M05, M19 := M19);												
		ELSE
			(* Get current axis specifc technology data *)			
			M_HandleTechnoAx(ADR(gpAx[nHliAxisIdx]^.techno_unit_std_sync[nLoop]), M03 := M03, M04 := M04, M05 := M05, M19 := M19);		
		END_IF																	
	END_FOR	
END_IF

IF nOpenTechnoCountLate > 0 THEN
	FOR nLoop := 0 TO nTechFctMaxIdxLate DO
		(* Depending on the source determined by parameter 'bIsChannelSpecific', the		*)
		(* channel or axis specific section of the HLI will be examined.					*)
		IF bIsChannelSpecific THEN			
			M_HandleTechnoCh(ADR(gpCh[nHliChannelIdx]^.techno_unit_late_sync[nLoop]), M03 := M03, M04 := M04, M05 := M05, M19 := M19);						
		ELSE
			(* Get current axis specifc technology data *)			
			M_HandleTechnoAx(ADR(gpAx[nHliAxisIdx]^.techno_unit_late_sync[nLoop]), M03 := M03, M04 := M04, M05 := M05, M19 := M19);	
		END_IF																	
	END_FOR	
END_IF
END_ACTION

METHOD PROTECTED M_HandleTechnoAx
VAR_INPUT
	pActTechnoUnit:	POINTER TO TECHNO_UNIT_AX;	
END_VAR
VAR_IN_OUT
	/// Raises if the cnc program encounters a M03 for the relevant spindle. Reset this for acknowledge 
	M03: BOOL;
	/// Raises if the cnc program encounters a M04 for the relevant spindle. Reset this for acknowledge 
	M04: BOOL;
	/// Raises if the cnc program encounters a M05 for the relevant spindle. Reset this for acknowledge 
	M05: BOOL;
	/// Raises if the cnc program encounters a M19 for the relevant spindle. Reset this for acknowledge 
	M19: BOOL;
END_VAR
		
		(* Check request *)
		IF pActTechnoUnit^.please_rw AND
		   NOT pActTechnoUnit^.done_w
		THEN
			CASE UINT_TO_UDINT(pActTechnoUnit^.fkt_ctrl_r) OF
		     (* -------------------------------------------------------------------------- *)
			 (* Handle M function *)
			 HLI_INTF_M_FKT:
				pMProcess					:= ADR(pActTechnoUnit^.attribut_r.data[0]);
				
				IF (pMProcess > 0) AND bHandleGearChange THEN
					CASE pMProcess^.nr OF
					 40:	M_ManageAcknowledgement(ADR(M40_Internal), pM40, ADR(bAcknowledge));
					 41:	M_ManageAcknowledgement(ADR(M41_Internal), pM41, ADR(bAcknowledge));
					 42:	M_ManageAcknowledgement(ADR(M42_Internal), pM42, ADR(bAcknowledge));
					 43:	M_ManageAcknowledgement(ADR(M43_Internal), pM43, ADR(bAcknowledge));
					 44:	M_ManageAcknowledgement(ADR(M44_Internal), pM44, ADR(bAcknowledge));
					 45:	M_ManageAcknowledgement(ADR(M45_Internal), pM45, ADR(bAcknowledge));
					END_CASE
				END_IF
				
			 (* -------------------------------------------------------------------------- *)
			 (* Handle S function *)
			 HLI_INTF_SPINDEL:
				pSProcess					:= ADR(pActTechnoUnit^.attribut_r.data[0]);
				
				(* If we are working with spindle functions provided by the channel 		*)
				(* specific section of the HLI the logical axis number transmitted from the *)
				(* CNC must fit the one given in parameter 'nLogAxisNoChannelSpecific'!					*)												
				IF bIsChannelSpecific AND (UINT_TO_INT(pSProcess^.log_achs_nr) <> nLogAxisNoChannelSpecific) THEN
					RETURN;
				END_IF
	
				CASE pSProcess^.move_cmd OF
				 (* ----------------------------------------------------------------------- *)
				 0: (* M19 *)
					IF (pSProcess^.pos_cmd = 19) AND
					   NOT M19_Internal THEN
						nPosition			:= pSProcess^.pos;
						M19_Internal		:= TRUE;
						M19					:= TRUE;
					ELSE
						IF NOT M19 THEN
							M19_Internal	:= FALSE;
							bAcknowledge	:= TRUE;
						END_IF
					END_IF
	
				 (* ----------------------------------------------------------------------- *)
				 3: (* M03 *)
					nRevolution				:= pSProcess^.rev;
	
					IF NOT M03_Internal THEN
						M03_Internal		:= TRUE;
						M03					:= TRUE;
					ELSE
						IF NOT M03 THEN
							M03_Internal	:= FALSE;
							bAcknowledge	:= TRUE;
						END_IF
					END_IF
	
				 (* ----------------------------------------------------------------------- *)
				 4: (* M04 *)
					nRevolution				:= pSProcess^.rev;
	
					IF NOT M04_Internal THEN
						M04_Internal		:= TRUE;
						M04					:= TRUE;
					ELSE
						IF NOT M04 THEN
							M04_Internal	:= FALSE;
							bAcknowledge	:= TRUE;
						END_IF
					END_IF
	
				 (* ----------------------------------------------------------------------- *)
				 5: (* M05 *)
					IF NOT M05_Internal THEN
						M05_Internal		:= TRUE;
						M05					:= TRUE;
					ELSE
						IF NOT M05 THEN
							M05_Internal	:= FALSE;
							bAcknowledge	:= TRUE;
						END_IF
					END_IF
	
				END_CASE
			END_CASE
	
			(* Handle acknowledgement *)
			IF bAcknowledge THEN
				bAcknowledge				:= FALSE;
				nRevolution					:= 0;
				nPosition					:= 0;
				pActTechnoUnit^.please_rw 	:= FALSE;
		   		pActTechnoUnit^.done_w		:= TRUE;
			END_IF
		END_IF
END_METHOD

METHOD PROTECTED M_HandleTechnoCh
VAR_INPUT
	pActTechnoUnit:	POINTER TO TECHNO_UNIT_CH;
END_VAR
VAR_IN_OUT
	/// Raises if the cnc program encounters a M03 for the relevant spindle. Reset this for acknowledge 
	M03: BOOL;
	/// Raises if the cnc program encounters a M04 for the relevant spindle. Reset this for acknowledge 
	M04: BOOL;
	/// Raises if the cnc program encounters a M05 for the relevant spindle. Reset this for acknowledge 
	M05: BOOL;
	/// Raises if the cnc program encounters a M19 for the relevant spindle. Reset this for acknowledge 
	M19: BOOL;
END_VAR
		
		(* Check request *)
		IF pActTechnoUnit^.please_rw AND
		   NOT pActTechnoUnit^.done_w
		THEN
			CASE UINT_TO_UDINT(pActTechnoUnit^.fkt_ctrl_r) OF
		     (* -------------------------------------------------------------------------- *)
			 (* Handle M function *)
			 HLI_INTF_M_FKT:
				pMProcess					:= ADR(pActTechnoUnit^.attribut_r.data[0]);
				
				IF (pMProcess > 0) AND bHandleGearChange THEN
					CASE pMProcess^.nr OF
					 40:	M_ManageAcknowledgement(ADR(M40_Internal), pM40, ADR(bAcknowledge));
					 41:	M_ManageAcknowledgement(ADR(M41_Internal), pM41, ADR(bAcknowledge));
					 42:	M_ManageAcknowledgement(ADR(M42_Internal), pM42, ADR(bAcknowledge));
					 43:	M_ManageAcknowledgement(ADR(M43_Internal), pM43, ADR(bAcknowledge));
					 44:	M_ManageAcknowledgement(ADR(M44_Internal), pM44, ADR(bAcknowledge));
					 45:	M_ManageAcknowledgement(ADR(M45_Internal), pM45, ADR(bAcknowledge));
					END_CASE
				END_IF
				
			 (* -------------------------------------------------------------------------- *)
			 (* Handle S function *)
			 HLI_INTF_SPINDEL:
				pSProcess					:= ADR(pActTechnoUnit^.attribut_r.data[0]);
				
				(* If we are working with spindle functions provided by the channel 		*)
				(* specific section of the HLI the logical axis number transmitted from the *)
				(* CNC must fit the one given in parameter 'nLogAxisNoChannelSpecific'!					*)												
				IF bIsChannelSpecific AND (UINT_TO_INT(pSProcess^.log_achs_nr) <> nLogAxisNoChannelSpecific) THEN
					RETURN;
				END_IF
	
				CASE pSProcess^.move_cmd OF
				 (* ----------------------------------------------------------------------- *)
				 0: (* M19 *)
					IF (pSProcess^.pos_cmd = 19) AND
					   NOT M19_Internal THEN
						nPosition			:= pSProcess^.pos;
						M19_Internal		:= TRUE;
						M19					:= TRUE;
					ELSE
						IF NOT M19 THEN
							M19_Internal	:= FALSE;
							bAcknowledge	:= TRUE;
						END_IF
					END_IF
	
				 (* ----------------------------------------------------------------------- *)
				 3: (* M03 *)
					nRevolution				:= pSProcess^.rev;
	
					IF NOT M03_Internal THEN
						M03_Internal		:= TRUE;
						M03					:= TRUE;
					ELSE
						IF NOT M03 THEN
							M03_Internal	:= FALSE;
							bAcknowledge	:= TRUE;
						END_IF
					END_IF
	
				 (* ----------------------------------------------------------------------- *)
				 4: (* M04 *)
					nRevolution				:= pSProcess^.rev;
	
					IF NOT M04_Internal THEN
						M04_Internal		:= TRUE;
						M04					:= TRUE;
					ELSE
						IF NOT M04 THEN
							M04_Internal	:= FALSE;
							bAcknowledge	:= TRUE;
						END_IF
					END_IF
	
				 (* ----------------------------------------------------------------------- *)
				 5: (* M05 *)
					IF NOT M05_Internal THEN
						M05_Internal		:= TRUE;
						M05					:= TRUE;
					ELSE
						IF NOT M05 THEN
							M05_Internal	:= FALSE;
							bAcknowledge	:= TRUE;
						END_IF
					END_IF
	
				END_CASE
			END_CASE
	
			(* Handle acknowledgement *)
			IF bAcknowledge THEN
				bAcknowledge				:= FALSE;
				nRevolution					:= 0;
				nPosition					:= 0;
				pActTechnoUnit^.please_rw 	:= FALSE;
		   		pActTechnoUnit^.done_w		:= TRUE;
			END_IF
		END_IF
END_METHOD

{attribute 'object_name' := 'M_ManageAcknowledgement'}
METHOD PRIVATE M_ManageAcknowledgement
VAR_INPUT
	pInternal: POINTER TO BOOL;
	pPublic: POINTER TO BOOL;
	pAcknowledgement: POINTER TO BOOL;
END_VAR
IF NOT pInternal^ THEN
	pInternal^			:= TRUE;
	pPublic^			:= TRUE;	
ELSIF NOT pPublic^ THEN
	pInternal^			:= FALSE;
	pAcknowledgement^	:= TRUE;
END_IF
END_METHOD

END_FUNCTION_BLOCK

// CNC/3 Control/HLI3_HandleSpindleTechnoGearchange
FUNCTION_BLOCK HLI3_HandleSpindleTechnoGearchange EXTENDS HLI3_HandleSpindleTechno
VAR_INPUT
END_VAR
VAR_OUTPUT
END_VAR
VAR_IN_OUT
		/// Raises if the cnc program encounters a M40 for the relevant spindle. Reset this for acknowledge 
	M40: BOOL;
	/// Raises if the cnc program encounters a M41 for the relevant spindle. Reset this for acknowledge 
	M41: BOOL;
	/// Raises if the cnc program encounters a M42 for the relevant spindle. Reset this for acknowledge 
	M42: BOOL;
	/// Raises if the cnc program encounters a M43 for the relevant spindle. Reset this for acknowledge 
	M43: BOOL;
	/// Raises if the cnc program encounters a M44 for the relevant spindle. Reset this for acknowledge 
	M44: BOOL;
	/// Raises if the cnc program encounters a M45 for the relevant spindle. Reset this for acknowledge 
	M45: BOOL;	
END_VAR
VAR
END_VAR

(* Date:	15/03/05																	*)
(* Author:	MiB																			*)
(* Rev:		1.0																			*)
(* ------------------------------------------------------------------------------------ *)
(* Desc 	Handling of spindle gear change M functions M40 - M45.						*)
(*			extends HLI3_SpindleTechno													*)
(*			overwrites the internal pointers to M40..M45 to VAR_IN_OUT					*)


SUPER^.pM40 := ADR(M40);
SUPER^.pM41 := ADR(M41);
SUPER^.pM42 := ADR(M42);
SUPER^.pM43 := ADR(M43);
SUPER^.pM44 := ADR(M44);
SUPER^.pM45 := ADR(M45);

A_HandleTechno();

END_FUNCTION_BLOCK

// CNC/3 Control/HLI3_SetAxisGantryOn
FUNCTION HLI3_SetAxisGantryOn : BOOL
VAR_INPUT
	nHliAxisIdx: INT;
	bEnable: BOOL;
END_VAR

(****************************************************************************************)
(* POU:		HLI_SetAxisGantryOn                      									*)
(* Type:	Function																	*)
(* Author: 	HR																			*)
(* Date: 	11/01/24																	*)
(* Rev.: 	1.0																			*)
(* ------------------------------------------------------------------------------------ *)
(* Desc:	Enables the axis specific control unit for driving out the gantry			*)
(*			difference. The actual movement is triggered by the input 'bEnable'.		*)
(*			The current axis has to be a gantry slave. That means:						*)
(*				+ It is not attached to a channel										*)
(*				+ kenngr.achs_mode		0x2000n		(where n specifies the axis type)	*)
(*				+ kenngr.gantry_ax_nr	1			(e. g. axis no. of gantry master)	*)
(*				+ kenngr.gantry_offset  10000		(e. g. difference to be driven out)	*)
(*				+ kenngr.gantry_vb_korr	20000		(e. g. velocity for driving out)	*)
(****************************************************************************************)

(* Check specified logical axis no first *)
IF NOT HLI3_CheckAxisValid(nHliAxisIdx := nHliAxisIdx) THEN
	HLI3_SetAxisGantryOn := FALSE;
	RETURN;
END_IF

gpAx[nHliAxisIdx]^.lr_mc_control.gantry_on.enable_w	:= TRUE;
gpAx[nHliAxisIdx]^.lr_mc_control.gantry_on.command_w	:= bEnable;
HLI3_SetAxisGantryOn	:= TRUE;

END_FUNCTION

// CNC/3 Control/HLI3_SetAxisReferencePosition
FUNCTION HLI3_SetAxisReferencePosition : BOOL
VAR_INPUT
	bSetRefpos: BOOL;
	nHliAxisIdx: INT;
END_VAR

(* ========================================================= *)
(*    FUN: HLI_SetAxisReferenceposition                      *)
(* --------------------------------------------------------- *)
(*   Desc:                                                   *)
(* Author: HR                                                *)
(*   Date: 09.11.2010                                        *)
(*   Rev.: 1.0                                               *)
(* ========================================================= *)
HLI3_SetAxisReferencePosition := FALSE;

IF NOT HLI3_CheckAxisValid(nHliAxisIdx := nHliAxisIdx) THEN	
	RETURN;
END_IF

(* set reference position *)
gpAx[nHliAxisIdx]^.lr_mc_control.set_reference_position.command_w := bSetRefpos;
HLI3_SetAxisReferencePosition := TRUE;

END_FUNCTION

// CNC/3 Control/HLI3_SetAxisSpindleStopAtProgramEnd
FUNCTION_BLOCK HLI3_SetAxisSpindleStopAtProgramEnd
VAR_INPUT
	bExecute: BOOL;
	bSpindelStopAtProgramEnd: BOOL;
	nHliAxisIdx: INT;
END_VAR
VAR_OUTPUT
	bBusy: BOOL;
END_VAR
VAR
	/// Index of axis specific HLI area 
	nHliAxIfcIdx: INT;
	nState: INT;
	fbRTrigExecute: R_TRIG;
END_VAR

(****************************************************************************************)
(* POU:		HLI_SetAxisSpindleStopAtProgramEnd                      					*)
(* Type:		FB																		*)
(* Author: 	HR                                              							*)
(* Date: 	24.01.11																	*)
(* Rev.: 	1.0                                               							*)
(* ------------------------------------------------------------------------------------ *)
(* Desc:	Check wether the axis specified by input 'nLogAxisNo' is a spindle and 		*)
(*			(re-) sets (depending on the state of input 'bSpindelStopAtProgramEnd') 	*)
(*			the spindle stop feature on the HLI.										*)
(****************************************************************************************)

(****************************************************************************************)
(*								Check logical axis no									*)
(****************************************************************************************)
IF NOT HLI3_CheckAxisValid(nHliAxisIdx := nHliAxisIdx) THEN	
	RETURN;
END_IF
(****************************************************************************************)
(*									Build trigger										*)
(****************************************************************************************)
fbRTrigExecute
	(CLK := bExecute);

(****************************************************************************************)
(*								   (Re-)set sequence									*)
(****************************************************************************************)
CASE nState OF
 (* ----------------------------------------------------------------------------------- *)
 0: (* INIT STATE  *)
  	bBusy			:= FALSE;

	IF fbRTrigExecute.Q THEN
		bBusy		:= TRUE;
		nState		:= 10;
	END_IF

 (* ----------------------------------------------------------------------------------- *)
 10: (* ENABLE THE CONTROL UNIT IF THE AXIS IS A SPINDLE *)

	IF gpAx[nHliAxisIdx]^.ipo_state.spindle_axis_r THEN
		gpAx[nHliAxisIdx]^.ipo_mc_control.spdl_stop_at_prog_end.enable_w := TRUE;
		nState 		:= 20;
	ELSE
		nState 		:= 0;
	END_IF

 (* ---------------------------------------------------------------------------------- *)
 20: (* (RE-) SET SPINDLE STOP FUNCTION *)
	gpAx[nHliAxisIdx]^.ipo_mc_control.spdl_stop_at_prog_end.command_w := bSpindelStopAtProgramEnd;
	nState 			:= 0;
END_CASE

END_FUNCTION_BLOCK

// CNC/3 Control/HLI3_SetAxisTrackingOperation
FUNCTION HLI3_SetAxisTrackingOperation : BOOL
VAR_INPUT
	nHliAxisIdx: INT;
	bPLCAxisEnable: BOOL;
END_VAR

(* ========================================================= *)
(*    FUN: HLI_SetAxisTrackingOperation                      *)
(* --------------------------------------------------------- *)
(*   Desc:                                                   *)
(*   Author: TV                                              *)
(*   Date: 15.09.2006                                        *)
(*   Rev.: 1.0                                               *)
(*         1.1 13.08.2013 Nachführbetrieb nicht bei Achsfehler einschalten *)
(* ========================================================= *)

IF NOT HLI3_CheckAxisValid(nHliAxisIdx := nHliAxisIdx) THEN	
	HLI3_SetAxisTrackingOperation := FALSE;
	RETURN;
END_IF

(* tracking operation (follow up) on / off *)
IF NOT bPLCAxisEnable THEN
	gpAx[nHliAxisIdx]^.lr_mc_control.follow_up.command_w := TRUE;
		HLI3_SetAxisTrackingOperation := TRUE;
ELSE
	gpAx[nHliAxisIdx]^.lr_mc_control.follow_up.command_w := FALSE;
		HLI3_SetAxisTrackingOperation := FALSE;
END_IF

END_FUNCTION

